// POUs/Functions/Gauges/Interfaces/FB_Gauge_Interface
(* This function block is created for interface devices between different PLC*)
(* Not all the Variables in the original structure is required, just few signals *)
(* They have to be linked to the custom created variables on the EL6692/5 primary side*)
FUNCTION_BLOCK FB_Gauge_Interface
VAR_INPUT
END_VAR
VAR_OUTPUT
	{attribute 'pytmc' := 'pv:'}
	VG : ST_VG;
END_VAR
VAR
	i_rPRESS AT%I*: REAL;  
	i_xAT_VAC AT%I*: BOOL;
	i_xPRESS_OK AT%I*: BOOL;
	
END_VAR

(* This function block is created for interface devices between different PLC*)
(* Not all the Variables in the original structure is required, just few signals *)
(* They have to be linked to the custom created variables on the EL6692/5 primary side*)

VG.rPRESS := i_rPRESS;
VG.xAT_VAC := i_xAT_VAC;
VG.xPRESS_OK := i_xPRESS_OK;

END_FUNCTION_BLOCK

// POUs/Functions/Gauges/Interfaces/FB_GaugeModbus
FUNCTION_BLOCK FB_GaugeModbus EXTENDS FB_GaugeBase
VAR_INPUT
	IP: STRING;	//IP of Legacy PLC
    nMBAddr	:WORD; //Start address of the Register Memory
	iBitOffset:INT :=0; // must be smaller than 32
	tTimeout :TIME:= T#1s;
END_VAR
VAR_OUTPUT
	VG: ST_VG;
	xNoPLCResponse: BOOL;
END_VAR
VAR
	fbPLCInputCoilsRx	:	FB_MBReadInputs;// (Modbus function 2)
	i_PLC_nBits	:	ARRAY [1..4] OF BYTE;
	ftReset	: F_TRIG; 
	tonRetry : TON;
	ErrCount:INT :=0;
	iIndex :INT;
	iBit:INT;
END_VAR
VAR CONSTANT
    nZero : INT := 0;
	nOne : INT := 1;
	nTwo : INT := 2;
	nThree : INT := 3;
	nFour : INT := 4;
	nFive : INT := 5;
	nSix : INT := 6;
	nSeven : INT := 7;
END_VAR

A_ReadMB();

ACTION A_ReadMB:
(*Credit to Alex Wallace*)
(* Modbus Info for Koyo
Modbus Addresses for
Koyo DL05/06/240/250/260/430/440/450 PLCs
PLC Memory Type		| Modbus start address Decimal (octal) | Function codes
Inputs (X)			  2048 (04000)							2
Special Relays (SP)	  3072 (06000)							2
Outputs (Y)			  2048 (04000)							1, 5, 15
Control Relays (C)	  3072 (06000)							1, 5, 15
Timer Contacts (T)	  6144 (014000)							1, 5, 15
Counter Contacts (CT) 6400 (014400)							1, 5, 15
Stage Status Bits (S) 6144 (012000)							1, 5, 15
*)

// Retry after some time
tonRetry.IN := NOT fbPLCInputCoilsRx.bBusy;
tonRetry.PT := T#10S;
tonRetry();

ftReset(CLK:=fbPLCInputCoilsRx.bBusy);
fbPLCInputCoilsRx.bExecute := ftReset.Q OR tonRetry.Q;

fbPLCInputCoilsRx(sIPAddr:=IP, nTCPPort:=502, nQuantity:=32, nMBAddr:=nMBAddr, cbLength:=SIZEOF(i_PLC_nBits),  pDestAddr:=ADR(i_PLC_nBits), tTimeout:=tTimeout);
//if there's a modbus error, set all incoming bits to zero
IF fbPLCInputCoilsRx.bError THEN
	i_PLC_nBits[1].0 := 0;
	i_PLC_nBits[1].1 := 0;
	i_PLC_nBits[1].2 := 0;
	i_PLC_nBits[1].3 := 0;
	i_PLC_nBits[1].4 := 0;
	i_PLC_nBits[1].5 := 0;
	i_PLC_nBits[1].6 := 0;
	i_PLC_nBits[1].7 := 0;
	i_PLC_nBits[2].0 := 0;
	i_PLC_nBits[2].1 := 0;
	i_PLC_nBits[2].2 := 0;
	i_PLC_nBits[2].3 := 0;
	i_PLC_nBits[2].4 := 0;
	i_PLC_nBits[2].5 := 0;
	i_PLC_nBits[2].6 := 0;
	i_PLC_nBits[2].7 := 0;
	VG.xPRESS_OK := FALSE;
	xNoPLCResponse:= TRUE;	
ELSIF NOT ftReset.Q AND fbPLCInputCoilsRx.cbRead > 0 THEN
	xNoPLCResponse:= FALSE;
	VG.rPRESS := 1E-8;
	iIndex:= REAL_TO_INT(iBitOffset/8);
	iBit:= (24 MOD 10);
	VG.xPRESS_OK := M_GetBit(iIndex,iBit);
	fbPLCInputCoilsRx.bExecute :=False;
ELSIF (*ftReset.Q*) NOT (fbPLCInputCoilsRx.bExecute) AND fbPLCInputCoilsRx.cbRead = 0 THEN
	xNoPLCResponse:= TRUE;		
END_IF

// Log Action
tAction(CLK:=   fbPLCInputCoilsRx.bError or xNoPLCResponse);
IF tAction.Q THEN 
ErrCount:= ErrCount+1; 
fbLogger(sMsg:='Modbus read error', eSevr:=TcEventSeverity.Critical);
END_IF
END_ACTION

METHOD M_GetBit : BOOL
VAR_INPUT
	iIndex:INT;
	iBit:INT;
END_VAR
Case iBit OF
	nZero: 
		M_GetBit:=i_PLC_nBits[iIndex].nZero;
	nOne: 
		M_GetBit:=i_PLC_nBits[iIndex].nOne;
	nTwo: 
		M_GetBit:=i_PLC_nBits[iIndex].nTwo;
	nThree: 
		M_GetBit:=i_PLC_nBits[iIndex].nThree;
	nFour: 
		M_GetBit:=i_PLC_nBits[iIndex].nFour;
	nFive: 
		M_GetBit:=i_PLC_nBits[iIndex].nFive;
	nSix: 
		M_GetBit:=i_PLC_nBits[iIndex].nSix;
	nSeven: 
		M_GetBit:=i_PLC_nBits[iIndex].nSeven;
END_CASE
END_METHOD

END_FUNCTION_BLOCK

// POUs/Functions/Gauges/Interfaces/FB_TGCC_ADS
(* This function block is created for interface devices between different PLC*)
(* Not all the Variables in the original structure is required, just few signals *)
(* The variable values are read via ADS using the symbol name*)
FUNCTION_BLOCK FB_TGCC_ADS Extends FB_ADS
VAR_INPUT
	sNetId : String; //NetID of the Destination PLC controller
	nPort : uint; // port number
	sVarName : string;// the variable name of the declared gauge function block.
	iWatchdog:UDINT;//The watchdog variable name written to by the remote plc
END_VAR
VAR_OUTPUT
	{attribute 'pytmc' := 'pv:'}
	IG : ST_VG;
	bError: BOOL;
END_VAR
VAR
	fb_CheckWatchdog: FB_CheckWatchdog;
	fb_Read_VG: FB_ReadAdsSymByName;
	ftReset: F_TRIG;
	xFirstPass: BOOL:= true;
END_VAR


ftReset(CLK:= fb_Read_VG.bBusy OR xFirstPass);
xFirstPass := false;
(*calling ADS read function*)

//IG.xPRESS_OK := false;	

fb_Read_VG(
	bRead:=ftReset.Q , 
	sNetId:= sNetId, 
	nPort:= nPort, 
	sVarName:= CONCAT(sVarName,'.IG'), 
	nDestAddr:= ADR(IG), 
	nLen:= SIZEOF(IG), 
	tTimeout:= , 
	eComMode:=eAdsComModeFastCom , 
	bBusy=> , 
	bError=> , 
	nErrorId=> );	
	

(*Error*)
fb_CheckWatchdog(
	bEnable:= TRUE, 
	tWatchdogTime:= T#900ms, 
	nCnt:= iWatchdog , 
	bWatchdog=> , 
	nLastCnt=> );
	
bError:= fb_Read_VG.bError OR fb_CheckWatchdog.bWatchdog;
tErrorPresent(CLK:=bError);

IF (fb_Read_VG.bError OR fb_CheckWatchdog.bWatchdog) THEN
IG.xPRESS_OK := FALSE;
END_IF;

(*Logger*)
ACT_Logger();

ACTION ACT_Logger:
IF tErrorPresent.Q THEN
 IF(fb_Read_VG.bError) THEN fbLogger(sMsg:='ADS Read Error', eSevr:=TcEventSeverity.Critical); END_IF;
 IF(fb_CheckWatchdog.bWatchdog) THEN fbLogger(sMsg:='ADS Watchdog Error', eSevr:=TcEventSeverity.Critical); END_IF;
END_IF
END_ACTION

END_FUNCTION_BLOCK

// POUs/Functions/Gauges/FB_972
{attribute 'no_check'}
FUNCTION_BLOCK FB_972  EXTENDS FB_GaugeBase
VAR_INPUT
END_VAR
VAR_OUTPUT
	{attribute 'pytmc' := '
    pv: 
	'}
	PG	: ST_VG;
END_VAR
VAR_IN_OUT
	
END_VAR
VAR
	rV : REAL;
	iTermBits: UINT := 32767 ; // The terminal's maximum value in bits
	(*IO*)
	i_iPRESS_R AT%I* :INT; // input Pressure // Link to analog Input
END_VAR

(* Standard MKS 9XX series conversion *)
(* works for 972 and 925 *)
// no div by zero
If (iTermBits=0) THEN iTermBits := 32767;END_IF
rV := 10*INT_TO_REAL(PG.i_iPRESS_R)/iTermBits;

IF rV > 1 THEN
	PG.rPRESS := LREAL_TO_REAL(EXPT(10, 2*rV-11));
	PG.xPRESS_OK := TRUE;
	PG.eState := Valid; //Press OK
ELSE
	PG.xPRESS_OK := FALSE;
	PG.eState := OoR;
END_IF



(* Soft IO Mapping*)
ACT_IO();

ACTION ACT_IO:
PG.i_iPRESS_R :=i_iPRESS_R;
END_ACTION

METHOD M_SetBits : BOOL
VAR_INPUT
	TermBits : UINT; // The terminal's maximum value in bits
END_VAR
This^.iTermBits := TermBits;
END_METHOD

END_FUNCTION_BLOCK

// POUs/Functions/Gauges/FB_9XX
(* Standard MKS 9XX series conversion *)
(* works for 925 *)
FUNCTION_BLOCK FB_9XX EXTENDS FB_GaugeBase
VAR_INPUT
END_VAR
VAR_OUTPUT
	{attribute 'pytmc' := '
    pv: 
	'}
	PG	: ST_VG;
END_VAR
VAR_IN_OUT
END_VAR
VAR
	rV : REAL;
	fbGaugeState : FB_PressureState;
	rMaxPressure	:	REAL := 760; //Torr
	rMinPressure	:	REAL := 1E-5; //Torr
	(*Default set point 50 mT*)
	rVAC_SP: REAL := 5E-2;
	iTermBits: UINT := 30518 ; // The terminal's maximum value in bits default el3174 as per vacuum architecture
	(*IO*)
	i_iPRESS_R AT%I* :INT; // input Pressure // Link to analog Input
END_VAR

(* Standard MKS 9XX series conversion *)
(* works for 972 and 925 *)

//Default setpoint 50 mT
IF PG.rVAC_SP = 0 THEN
	PG.rVAC_SP := rVAC_SP;
END_IF
// check no div by zero
If (iTermBits=0) THEN iTermBits := 30518;END_IF
rV := 10*INT_TO_REAL(PG.i_iPRESS_R)/iTermBits;

IF rV >= 0.99 THEN
	IF rV >= 0.99 AND rV <= 1 THEN
		PG.rPRESS := 1E-5;
	ELSE
		PG.rPRESS := LREAL_TO_REAL(EXPT(10, rV-6));
	END_IF
	PG.xPRESS_OK := TRUE;
	PG.eState := Valid;
ELSE
	PG.xPRESS_OK := FALSE;
	IF (rV = 0) THEN PG.eState := GaugeDisconnected;
		ELSE  PG.eState := PressInvalid;
	END_IF
END_IF

(* Setpoint evaluation *)
PG.xAT_VAC := PG.xPRESS_OK AND (PG.rPRESS < PG.rVAC_SP);


(*Logger*)
ACT_Logger();
(*Soft IO Mapping*)
ACT_IO();

ACTION ACT_IO:
PG.i_iPRESS_R :=i_iPRESS_R;
END_ACTION

ACTION ACT_Logger:

//STATE Logger  
IF ePrevState <> PG.eState THEN
	  CASE PG.eState OF
		ValidHi:
			fbLogger(sMsg:='Gauge pressure valid high.', eSevr:=TcEventSeverity.Info);
		ValidLo:
			fbLogger(sMsg:='Gauge pressure valid low.', eSevr:=TcEventSeverity.Info);
		Valid:
			fbLogger(sMsg:='Gauge pressure valid.', eSevr:=TcEventSeverity.Info);
  		GaugeDisconnected:
			fbLogger(sMsg:='Gauge Disconnected.', eSevr:=TcEventSeverity.Critical);
		PressInvalid:
			fbLogger(sMsg:='Gauge pressure invalid.', eSevr:=TcEventSeverity.Warning);
		OoR:
			fbLogger(sMsg:='Gauge pressure out of range.', eSevr:=TcEventSeverity.Warning);
		Starting:
			fbLogger(sMsg:='Gauge starting.', eSevr:=TcEventSeverity.Info);
	  END_CASE
	  ePrevState := PG.eState;  
  END_IF
END_ACTION

METHOD M_SetBits : BOOL
VAR_INPUT
	TermBits : UINT; // The terminal's maximum value in bits
END_VAR
This^.iTermBits := TermBits;
END_METHOD

END_FUNCTION_BLOCK

// POUs/Functions/Gauges/FB_CMR362
(* For Pfeiffer CMR 362 *)
FUNCTION_BLOCK FB_CMR362
VAR_INPUT
END_VAR
VAR_OUTPUT
		{attribute 'pytmc' := 'pv:'}
		PG : ST_VG;
END_VAR
VAR
	MinPressure: REAL := 7.5E-3; //Torr
	FullScale : REAL := 75.0 ; //Torr
	V : REAL;
	iTermBits: UINT := 32767 ; // The terminal's maximum value in bits
	(*IO*)
	i_iPRESS_R AT%I* :INT; // input Pressure // Link to analog Input
END_VAR


(* For Pfeiffer CMR 362 *)
(*Soft IO Mapping*)
ACT_IO();

(* Real-value calculation *)
If (iTermBits=0) THEN iTermBits := 32767;END_IF
V := 10*INT_TO_REAL(PG.i_iPRESS_R)/iTermBits;
	

IF V < 0.4 THEN

	PG.eState := GaugeDisconnected; //Most likely not connected

ELSIF V >= 0.4 AND V <= 1.0 THEN
	PG.rPRESS := MinPressure;
	PG.eState := ValidLo;

ELSIF V > 1 AND V <= 9.8 THEN

	PG.rPRESS := LREAL_TO_REAL((V-1)*0.125*FullScale);
	PG.eState := Valid;

ELSE
	
PG.eState := OoR; //Larger voltage, probably out of range?

END_IF


(* Pressure OK check *)
PG.xPRESS_OK := (PG.rPRESS >= MinPressure);

(*Soft IO Mapping*)
ACT_IO();

ACTION ACT_IO:
PG.i_iPRESS_R :=i_iPRESS_R;
END_ACTION

METHOD M_SetBits : BOOL
VAR_INPUT
	TermBits : UINT; // The terminal's maximum value in bits
END_VAR
This^.iTermBits := TermBits;
END_METHOD

END_FUNCTION_BLOCK

// POUs/Functions/Gauges/FB_GCM
(* For Baratron Pressure Gauge *)
(*The full-scale pressure times the ratio of the meas.
voltage to full-scale voltage (10V).
The minimum pressure is always going to be 5e-4 * F.S.V.*)
FUNCTION_BLOCK FB_GCM
VAR_IN_OUT

END_VAR
VAR_OUTPUT
	{attribute 'pytmc' := 'pv:'}
	PG	:	ST_VG;
END_VAR
VAR_INPUT
	i_rFULL_SCALE : REAL;
END_VAR
VAR
	rMinPressure: REAL;
	rHYST_PERC	:	REAL := 0.80;	// Hysteresis percentage
	rV	:REAL;
	iTermBits: UINT := 32767 ; // The terminal's maximum value in bits
	(*IO*)
	i_iPRESS_R AT%I* :INT; // input Pressure // Link to analog Input
END_VAR

(* Baratron Pressure Calc 
A. Wallace
2016-6-16
The full-scale pressure times the ratio of the meas.
voltage to full-scale voltage (10V).
The minimum pressure is always going to be 5e-4 * F.S.V.*)
PG.rFULL_SCALE := i_rFULL_SCALE;
rMinPressure := PG.rFULL_SCALE * 5E-4;

If (iTermBits=0) THEN iTermBits := 32767;END_IF
rV :=MAX((10*INT_TO_REAL(PG.i_iPRESS_R)/iTermBits),0);

PG.rPRESS := (PG.rFULL_SCALE/10)*rV;
IF PG.rPRESS > (rMinPressure)THEN
	PG.xPRESS_OK := TRUE;
ELSE
	PG.xPRESS_OK := FALSE;
END_IF

(*IO soft linking*)
ACT_IO();

ACTION ACT_IO:
PG.i_iPRESS_R :=i_iPRESS_R;
END_ACTION

METHOD M_SetBits : BOOL
VAR_INPUT
	TermBits : UINT; // The terminal's maximum value in bits
END_VAR
This^.iTermBits := TermBits;
END_METHOD

END_FUNCTION_BLOCK

// POUs/Functions/Gauges/FB_ITR90
(* This function block implements the Oerlikon Leybold IONVAC Hot Cathode ITR 90*)
FUNCTION_BLOCK FB_ITR90
VAR_INPUT
END_VAR
VAR_OUTPUT
	{attribute 'pytmc' := '
    pv: 
	'}
	PG : ST_VG;
END_VAR
VAR
	rV : REAL;	// input voltage
	rC: REAL := -0.125; // a constant in the manual (pressure unit dependent)
	rK: REAL := 1.0;// Calibration factor C (gas type dependent)
	iTermBits: UINT := 32767 ; // The terminal's maximum value in bits
	(*IO*)
	i_iPRESS_R AT%I* :INT; // input Pressure // Link to analog Input
END_VAR

(* This function block implements the Oerlikon Leybold IONVAC Hot Cathode ITR 90*)

(* Real-value calculation *)

rV := 10*INT_TO_REAL(PG.i_iPRESS_R)/iTermBits;	
PG.rPRESS := (LREAL_TO_REAL(EXPT(10,(rV-7.75)/0.75+rC))) * rK;


(* Pressure gauge State checks *)

//IF (rV <=9.7 ) AND (rV>=1) THEN
	//PG.eState := Valid; // normal
IF rV >= 0.5 AND rV <= 4.5 THEN
	PG.eState := ValidLo; //LO
ELSIF rV > 4.5 AND rV<= 9.9 THEN
	PG.eState := ValidHi; //HIGH
ELSIF rV < 0.5 THEN
	PG.eState := GaugeDisconnected; //not on
ELSE
	PG.eState := PressInvalid; //other fault - could be no gauge, controller powering up etc
END_IF



(* Pressure gauge OK checks *)
PG.xPRESS_OK := (rV <=9.9 ) AND (rV>=0.5);


(* Setpoint evaluation *)
PG.xAT_VAC := PG.xPRESS_OK AND PG.rPRESS < PG.rVAC_SP;


(*Soft IO Linking*)
ACT_IO();

ACTION ACT_IO:
PG.i_iPRESS_R :=i_iPRESS_R;
END_ACTION

METHOD M_SetBits : BOOL
VAR_INPUT
	TermBits : UINT; // The terminal's maximum value in bits
END_VAR
If (iTermBits=0) THEN iTermBits := 32767;END_IF
This^.iTermBits := TermBits;
END_METHOD

END_FUNCTION_BLOCK

// POUs/Functions/Gauges/FB_MKS_937A
(* 937A Logarithmic Output Conversion *)
(* 7-15-2015 *)
(* This function will read the pressure from any gauge on a 937A. *)
(* To be used when the specific device function block is not available *)
FUNCTION_BLOCK FB_MKS_937A
VAR_IN_OUT
	
END_VAR
VAR_INPUT
	PG	:	ST_VG := g_DummyVG; // Gauge Structure used to Interlock the ion gauges
END_VAR
VAR_OUTPUT
	{attribute 'pytmc' := 'pv: '}
	VG : ST_VG; // Vacuum Gauge Data Structure
END_VAR
VAR
	rV	:	REAL;
		(*IOs to be linked*)
	/// Controls and I/Os
	i_iPRESS_R AT %I* :INT; // input Pressure // Link to analog Input
	q_xHV_DIS AT %Q* : BOOL; // Disable Gauge High Voltage when True // 'TcLinkTo' (EL2794) ^Output
	
END_VAR

(* 937A Logarithmic Output Conversion *)
(* 7-15-2015 *)
(* This function will read the pressure from any gauge on a 937A. *)

rV := 10*INT_TO_REAL(VG.i_iPRESS_R)/32767;
VG.rPRESS := LREAL_TO_REAL(EXPT(10,rV/0.6-12));


(* Ion Gauge Protection Functions *)
(* If the PG pressure is greater than the VG.PRO_SP then the gauge is disabled *)
(* If the PG pressure is less than the VG.PRO_SP then the gauge is enabled *)
(* This FB also implements some hysteresis so the gauge doesn't have rapid power cycling while near the turn on boundary *)

IF PG.rPRESS < VG.rPRO_SP THEN

VG.q_xHV_DIS :=  NOT VG.xHV_SW;

ELSIF NOT VG.q_xHV_DIS THEN
	IF VG.rPRESS > VG.rPRO_SP + VG.rHYS_PR OR PG.rPRESS > VG.rPRO_SP + VG.rHYS_PR THEN
		VG.q_xHV_DIS := TRUE;
	END_IF
ELSE
	VG.q_xHV_DIS := TRUE;
END_IF


(* Pressure gauge OK checks *)
VG.xPRESS_OK := (rV <=9.6 ) AND (rV>=0.6); //legacy

IF (rV <=9.6 ) AND (rV>=0.6) THEN
	VG.eState := Valid; // normal
ELSIF rV >= 0.18 AND rV <= 0.22 THEN
	VG.eState := ValidLo; //LO
ELSIF rV >= 9.7 AND rV<= 9.9 THEN
	VG.eState := ValidHi; //HIGH
ELSIF rV < 0.18 THEN
	VG.eState := GaugeDisconnected; //not on
ELSE
	VG.eState := PressInvalid; //other fault - could be no gauge, controller powering up etc
END_IF

(* Setpoint evaluation *)
VG.xAT_VAC := (VG.eState =Valid) AND VG.rPRESS < VG.rVAC_SP;

(*Soft IO Linking*)
ACT_IO();

ACTION ACT_IO:
(*soft link inputs*)
VG.i_iPRESS_R:=	i_iPRESS_R; 

(*soft link outputs*)
q_xHV_DIS := VG.q_xHV_DIS;
END_ACTION

END_FUNCTION_BLOCK

// POUs/Functions/Gauges/FB_MKS_937B
(* 937B Logarithmic Output Conversion *)
(* 5-20-2016, Alex Wallace and Scott Stubbs *)
(* This function will read the pressure from any gauge on a 937B. *)
(* To be used when the specific device function block is not available *)
FUNCTION_BLOCK FB_MKS_937B
VAR_IN_OUT
			
END_VAR
VAR_INPUT
	PG	:	ST_VG := g_DummyVG; // Gauge Structure used to Interlock the ion gauges
END_VAR
VAR_OUTPUT
	{attribute 'pytmc' := 'pv: '}
	VG : ST_VG; // Vacuum Gauge Data Structure
	
	

END_VAR
VAR
	rV	:	REAL;
	
	
		(*IOs to be linked*)
	/// Controls and I/Os
	i_iPRESS_R AT %I* :INT; // input Pressure // Link to analog Input
	q_xHV_DIS AT %Q* : BOOL; // Disable Gauge High Voltage when True // 'TcLinkTo' (EL2794) ^Output
	
END_VAR

(* 937B Logarithmic Output Conversion *)
(* 5-20-2016, Alex Wallace and Scott Stubbs *)
(* This function will read the pressure from any gauge on a 937B. *)

rV := 10*INT_TO_REAL(VG.i_iPRESS_R)/32767;
VG.rPRESS := LREAL_TO_REAL(EXPT(10,(rV-7.2)/0.6));


(* Gauge Protection Functions *)
(* If the PG pressure is greater than the VG.PRO_SP then the gauge is disabled *)
(* If the PG pressure is less than the VG.PRO_SP then the gauge is enabled *)
(* This FB also implements some hysteresis so the gauge doesn't have rapid power cycling while near the turn on boundary *)

IF PG.rPRESS < VG.rPRO_SP THEN // might enable the gauge automatically, do we want that?

VG.q_xHV_DIS := NOT VG.xHV_SW;

ELSIF NOT VG.q_xHV_DIS THEN
	IF VG.rPRESS > VG.rPRO_SP + VG.rHYS_PR OR PG.rPRESS > VG.rPRO_SP + VG.rHYS_PR THEN
		VG.q_xHV_DIS := TRUE;
	END_IF
ELSE
	VG.q_xHV_DIS := TRUE;
END_IF


(* Pressure gauge OK checks *)
VG.xPRESS_OK := (rV <=9.6 ) AND (rV>=0.6);
(* Pressure gauge State checks *)
IF (rV <=9.7 ) AND (rV>=0.6) THEN
	VG.eState := Valid; // normal
ELSIF rV >= 0.18 AND rV <= 0.22 THEN
	VG.eState := ValidLo; //LO
ELSIF rV > 9.7 AND rV<= 9.9 THEN
	VG.eState := ValidHi; //HIGH
ELSIF rV < 0.18 THEN
	VG.eState := GaugeDisconnected; //not on
ELSE
	VG.eState := PressInvalid; //other fault - could be no gauge, controller powering up etc
END_IF

(* Setpoint evaluation *)
VG.xAT_VAC := (VG.eState =Valid) AND VG.rPRESS < VG.rVAC_SP;


(*Soft IO Linking*)
// check ethercat Diagnostics
ACT_IO();

ACTION ACT_IO:
(*soft link inputs*)
VG.i_iPRESS_R:=	i_iPRESS_R; 

(*soft link outputs*)
q_xHV_DIS := VG.q_xHV_DIS;
END_ACTION

END_FUNCTION_BLOCK

// POUs/Functions/Gauges/FB_MKS275
(* This function block is used to provide protection and automatic turn on of ion gauges,
 it also manages the turn on of the AT_VAC boolean, and checks to make sure the pressure is good *)
(* For MKS 275 mini-convectron *)
{attribute 'no_check'}
FUNCTION_BLOCK FB_MKS275 EXTENDS FB_GaugeBase
VAR_IN_OUT

END_VAR
VAR_INPUT
END_VAR

VAR_OUTPUT
	{attribute 'pytmc' := '
    pv: 
	'}
	PG : ST_VG;
END_VAR
VAR
	V : REAL;
	iTermBits: UINT := 32767 ; // The terminal's maximum value in bits
	Vlowest: REAL := 10;
	(*IO*)
	i_iPRESS_R AT%I* :INT; // input Pressure // Link to analog Input
END_VAR

VAR CONSTANT
	MinPressure: REAL := 1E-4;
	rDeadband : REAL :=0.05;
	rValidLoBoundary	:	REAL := 0.375; //  0.375V as per manual page 27
	rValidHiBoundary	:	REAL := 5.659;// 5.534; // manual page 27
	rDisconnectedBoundary	:	REAL := 0.3;
END_VAR

(* This function block is used to provide protection and automatic turn on of ion gauges,
 it also manages the turn on of the AT_VAC boolean, and checks to make sure the pressure is good *)
(* For MKS 275 mini-convectron *)

//Default setpoint 50 mT
IF PG.rVAC_SP = 0 THEN
	PG.rVAC_SP := 5E-2;
END_IF

(* Real-value calculation *)
If (iTermBits=0) THEN iTermBits := 32767;END_IF
V := 10*INT_TO_REAL(PG.i_iPRESS_R)/iTermBits;	

Vlowest := MIN(V, Vlowest);

IF V > rDisconnectedBoundary AND V < rValidLoBoundary  THEN
	PG.rPRESS := MinPressure;
	PG.eState := ValidLo;
	
ELSIF V >= rValidLoBoundary AND V < rValidLoBoundary +rDeadband  THEN
	PG.rPRESS := MAX( MinPressure, LREAL_TO_REAL( -0.02585 + 0.03767*V + 0.04563*EXPT(V,2)+ 0.1151*EXPT(V,3) - 0.04158*EXPT(V,4)+ 0.008737*EXPT(V,5)) );
	PG.eState := ValidLo;
	
ELSIF V >= rValidLoBoundary AND V < 2.842 THEN
	PG.rPRESS := MAX( MinPressure, LREAL_TO_REAL( -0.02585 + 0.03767*V + 0.04563*EXPT(V,2)+ 0.1151*EXPT(V,3) - 0.04158*EXPT(V,4)+ 0.008737*EXPT(V,5)) );
	PG.eState := Valid;

ELSIF V >= 2.842 AND V < 4.945 THEN
	PG.rPRESS := LREAL_TO_REAL((0.1031-0.02322*V+0.07229*EXPT(V,2))/(1-0.3986*V+0.07438*EXPT(V,2)-0.006866*EXPT(V,3)));
	PG.eState := Valid;

ELSIF V >= 4.945 AND V < rValidHiBoundary THEN
	PG.rPRESS := LREAL_TO_REAL((100.624-20.5623*V)/(1-0.37679*V+0.0348656*EXPT(V,2)));
	PG.eState := ValidHi;

ELSIF V <= rDisconnectedBoundary THEN
	PG.eState := GaugeDisconnected; //Most likely not connected
	PG.rPRESS := -1;

ELSE
	PG.eState := OoR; //Larger voltage, probably out of range?
	PG.rPRESS := -1;
END_IF

(* Protection Functions *)
(* If the PG pressure is greater than the IG.PRO_SP then the gauge is disabled *)
(* If the PG pressure is less than the IG.PRO_SP then the gauge is enabled *)
(* This FB also implements some hysteresis so the gauge doesn't have rapid power cycling while near the turn on boundary *)

(* Pressure OK check *)
PG.xPRESS_OK := (PG.rPRESS >= MinPressure);

(* Setpoint evaluation *)
PG.xAT_VAC := PG.xPRESS_OK AND (PG.rPRESS<=PG.rVAC_SP);

(*Logger*)
ACT_Logger();

(*Soft IO Mapping *)
IO();

ACTION ACT_Logger:

//STATE Logger  
if (PG.xLog) THEN
	IF ePrevState <> PG.eState THEN
	  CASE PG.eState OF
		ValidHi:
			fbLogger(sMsg:='Gauge pressure valid high.', eSevr:=TcEventSeverity.Info);
		ValidLo:
			fbLogger(sMsg:='Gauge pressure valid low.', eSevr:=TcEventSeverity.Info);
		Valid:
			fbLogger(sMsg:='Gauge pressure valid.', eSevr:=TcEventSeverity.Info);
  		GaugeDisconnected:
			fbLogger(sMsg:='Gauge Disconnected.', eSevr:=TcEventSeverity.Critical);
		PressInvalid:
			fbLogger(sMsg:='Gauge pressure invalid.', eSevr:=TcEventSeverity.Warning);
		OoR:
			fbLogger(sMsg:='Gauge pressure out of range.', eSevr:=TcEventSeverity.Warning);
		Starting:
			fbLogger(sMsg:='Gauge starting.', eSevr:=TcEventSeverity.Info);
	  END_CASE
	  ePrevState := PG.eState;  
  END_IF 
END_IF
END_ACTION

ACTION IO:
PG.i_iPRESS_R :=i_iPRESS_R;
PG.sPath := sPath;
END_ACTION

METHOD M_SetBits : BOOL
VAR_INPUT
	TermBits : UINT; // The terminal's maximum value in bits
END_VAR
This^.iTermBits := TermBits;
END_METHOD

END_FUNCTION_BLOCK

// POUs/Functions/Gauges/FB_MKS317
(* This function is for the Pirani MKS 317 connected to a 937A/B *)
(* This function block is used to provide protection and automatic turn on of ion gauges,
 it also manages the turn on of the AT_VAC boolean, and checks to make sure the pressure is good *)

FUNCTION_BLOCK FB_MKS317 Extends FB_GaugeBase
VAR_IN_OUT
END_VAR
VAR_INPUT
	b937A :BOOL := FALSE; // True if this gauge is connected to MKS937A controller, False if connected to MKS937B controller
END_VAR
VAR_OUTPUT
	{attribute 'pytmc' := '
    pv: 
	'}
	PG : ST_VG;
END_VAR
VAR
	rV	:	REAL;

	(*IO*)
	i_iPRESS_R AT%I* :INT; // input Pressure // Link to analog Input
END_VAR

VAR CONSTANT
	rMinPressure: REAL := 1E-4;
	rDefaultVAC_SP: REAL :=5E-2; // Default 50 mT
	rDisconnectedBoundary	:	REAL := 0.10;
	rValidLoBoundary	:	REAL := 0.22;
	rValidBoundaryMin	:	REAL := 0.6;
	rValidHiBoundary	:	REAL := 9.7;
	rValidHiBoundaryMax	:	REAL := 9.9; 
	rNoSensorBoundary	:	REAL := 10;
END_VAR

(* 937B Logarithmic Output Conversion *)
(* 5-20-2016, Alex Wallace and Scott Stubbs *)
(* 09-28-2018, Margaret Ghaly *)
(* This function will read the pressure from any gauge on a 937B. *)

rV := 10*INT_TO_REAL(PG.i_iPRESS_R)/32767;
if (b937A) THEN
	PG.rPRESS := LREAL_TO_REAL(EXPT(10,((rV)/0.6)-12)); //manual page 61 MKS937A
	ELSE
	PG.rPRESS := LREAL_TO_REAL(EXPT(10,(rV-7.2)/0.6));	//manual page 73 MKS937B
END_IF


//Default setpoint 
IF PG.rVAC_SP = 0 THEN
	PG.rVAC_SP := rDefaultVAC_SP;
END_IF

IF (rV <=rValidHiBoundary ) AND (rV>=rValidBoundaryMin) THEN
	PG.eState := Valid; // normal
ELSIF rV >= rDisconnectedBoundary AND rV <= rValidLoBoundary THEN
	PG.eState := ValidLo; //LO
	PG.rPRESS := rMinPressure;
ELSIF rV > rValidHiBoundary AND rV<= rValidHiBoundaryMax THEN
	PG.eState := ValidHi; //HIGH
ELSIF rV < rDisconnectedBoundary THEN
	PG.eState := GaugeDisconnected; //not on
	PG.rPRESS := -1;
ELSE
	PG.eState := PressInvalid; //other fault - could be no gauge, controller powering up etc
	PG.rPRESS := -1;
END_IF

(* Pressure OK check *)
(* Pressure gauge OK checks *)
PG.xPRESS_OK := (rV <=rValidHiBoundary ) AND (rV>=rDisconnectedBoundary);
//PG.xPRESS_OK := (PG.rPRESS >= rMinPressure);

(* Setpoint evaluation *)
PG.xAT_VAC := (*(PG.eState =Valid)*) PG.xPRESS_OK AND PG.rPRESS <= PG.rVAC_SP;

(*Logger*)
ACT_Logger();

(*soft io*)
IO();

ACTION ACT_Logger:

//STATE Logger  
IF (PG.xLog) THEN
	IF ePrevState <> PG.eState THEN
		  CASE PG.eState OF
			ValidHi:
				fbLogger(sMsg:='Gauge pressure valid high.', eSevr:=TcEventSeverity.Info);
			ValidLo:
				fbLogger(sMsg:='Gauge pressure valid low.', eSevr:=TcEventSeverity.Info);
			Valid:
				fbLogger(sMsg:='Gauge pressure valid.', eSevr:=TcEventSeverity.Info);
			GaugeDisconnected:
				fbLogger(sMsg:='Gauge Disconnected.', eSevr:=TcEventSeverity.Critical);
			PressInvalid:
				fbLogger(sMsg:='Gauge pressure invalid.', eSevr:=TcEventSeverity.Warning);
			OoR:
				fbLogger(sMsg:='Gauge pressure out of range.', eSevr:=TcEventSeverity.Warning);
			Starting:
				fbLogger(sMsg:='Gauge starting.', eSevr:=TcEventSeverity.Info);
		  END_CASE
		  ePrevState := PG.eState;  
	  END_IF
 END_IF
END_ACTION

ACTION IO:
PG.i_iPRESS_R :=i_iPRESS_R;

PG.sPath := sPath;
END_ACTION

END_FUNCTION_BLOCK

// POUs/Functions/Gauges/FB_MKS392
(* This function block implements the MKS392 gauge*)
FUNCTION_BLOCK FB_MKS392
VAR_INPUT
END_VAR
VAR_OUTPUT
	{attribute 'pytmc' := '
    pv: 
	'}
	PG : ST_VG;
END_VAR
VAR
	rV : REAL;	// input voltage
	iTermBits: UINT := 32767 ; // The terminal's maximum value in bits
	(*IO*)
	i_iPRESS_R AT%I* :INT; // input Pressure // Link to analog Input
END_VAR

(* Real-value calculation *)
rV := 10*INT_TO_REAL(PG.i_iPRESS_R)/iTermBits;	
PG.rPRESS := (LREAL_TO_REAL(EXPT(10,(2*rV)-11)));


(* Pressure gauge State checks *)

IF rV >= 0.5 AND rV <= 3.5 THEN
	PG.eState := ValidLo; //LO
ELSIF rV > 3.5 AND rV<= 6.5 THEN
	PG.eState := ValidHi; //HIGH
ELSIF rV < 0.5 THEN
	PG.eState := GaugeDisconnected; //not on
ELSE
	PG.eState := PressInvalid; //other fault - could be no gauge, controller powering up etc
END_IF



(* Pressure gauge OK checks *)
PG.xPRESS_OK := (rV <=6.5 ) AND (rV>=0.5);


(* Setpoint evaluation *)
PG.xAT_VAC := PG.xPRESS_OK AND PG.rPRESS < PG.rVAC_SP;


(*Soft IO Linking*)
ACT_IO();

ACTION ACT_IO:
PG.i_iPRESS_R :=i_iPRESS_R;
END_ACTION

END_FUNCTION_BLOCK

// POUs/Functions/Gauges/FB_MKS422
(* This function is for the Cold Cathode MKS 422 connected to a 937A/B *)
(*This function provides ILK and Set Point Protection for the Cold Cathode*)
FUNCTION_BLOCK FB_MKS422 EXTENDS FB_GaugeBase
VAR_IN_OUT
		
END_VAR
VAR_INPUT
		PG	:	ST_VG; // Pirani Gauge Structure used to Interlock the Cold Cathode
		b937A :BOOL:=FALSE; // True if this gauge is connected to MKS937A controller, False if connected to MKS937B controller
END_VAR
VAR_OUTPUT
	{attribute 'pytmc' := '
    pv: 
	'}
	IG : ST_VG; // The Cold Cathode Data Structure
END_VAR
VAR
	rV	:	REAL;
	
	timer:TON;
	(*IOs to be linked*)
	/// Controls and I/Os
	i_iPRESS_R AT %I* :INT; // input Pressure // Link to analog Input
	q_xHV_DIS AT %Q* : BOOL := True; // Disable Gauge High Voltage when True // 'TcLinkTo' (EL2794) ^Output
END_VAR
VAR CONSTANT
	MinPressure: REAL := 1E-10;
	cDefaultPressure : REAL := 0;
END_VAR

(* 937B Logarithmic Output Conversion *)
(* 5-20-2016, Alex Wallace and Scott Stubbs *)
(* 09-28-2018, Margaret Ghaly *)
(* This function will read the pressure from any gauge on a 937B. *)

(*Soft IO Linking*)
IO();

(*Pressure readbacks*)
rV := 10*INT_TO_REAL(IG.i_iPRESS_R)/32767;
if (b937A) THEN
	IG.rPRESS := LREAL_TO_REAL(EXPT(10,((rV)/0.6)-12)); //manual page 61 MKS937A
	ELSE
	IG.rPRESS := LREAL_TO_REAL(EXPT(10,(rV-7.2)/0.6));	//manual page 73 MKS937B
END_IF

	

(* Pressure gauge State checks *)
IF (rV <=9.6 ) AND (rV>=0.6) THEN
	IG.eState := Valid; // normal
ELSIF rV >= 0.18 AND rV <= 0.22 THEN 
	IG.eState := ValidLo; //LO
ELSIF rV > 9.6 AND rV<= 9.9 THEN
	IG.eState := ValidHi; //HIGH
ELSIF rV < 0.18 THEN // 
	IG.eState := GaugeDisconnected; //not on
	IG.rPRESS :=cDefaultPressure;
ELSE
	IG.eState := PressInvalid; //other fault - could be no gauge, controller powering up etc
	IG.rPRESS :=cDefaultPressure;
END_IF


(* Ion Gauge Protection Functions *)
(* If the PG pressure is greater than the VG.PRO_SP then the gauge is disabled *)
(* If the PG pressure is less than the VG.PRO_SP then the gauge is enabled *)
(* This FB also implements some hysteresis so the gauge doesn't have rapid power cycling while near the turn on boundary *)

	IF (PG.rPRESS <= IG.rPRO_SP) THEN
		 IG.q_xHV_DIS := NOT IG.xHV_SW;
		 IG.xILKOk := TRUE;
	ELSIF NOT IG.q_xHV_DIS AND timer.Q THEN
		IF IG.rPRESS > (IG.rPRO_SP + IG.rHYS_PR) OR PG.rPRESS > (IG.rPRO_SP + IG.rHYS_PR) THEN
		IG.q_xHV_DIS := TRUE;
		IG.xHV_SW := FALSE;
		END_IF
	ELSE 
		IG.q_xHV_DIS := TRUE;
		IG.xHV_SW := FALSE;
		IG.xILKOk := FALSE;
 	END_IF
 


 
(* Pressure gauge OK checks *)
IG.xPRESS_OK := (rV <=9.6 ) AND (rV>=0.6);


(* Setpoint evaluation *)
IG.xAT_VAC := IG.xPRESS_OK AND IG.rPRESS < IG.rVAC_SP;


(*Logger*)
ACT_Logger();
(*Soft IO Linking*)
// check ethercat Diagnostics
IO();

timer(IN:= NOT IG.q_xHV_DIS, PT:= T#2s);

ACTION ACT_Logger:
// ILK logger
IF (IG.xLog) THEN
	IF NOT IG.xILKOk AND NOT IG.q_xHV_DIS THEN
			fbLogger(sMsg:='Lost external interlock while gauge was on.', eSevr:=TcEventSeverity.Critical);  	
	END_IF
	
	
	// Log Action
	tAction(CLK:=  IG.xHV_SW);
	IF tAction.Q THEN fbLogger(sMsg:='Ion gauge commanded to switch on', eSevr:=TcEventSeverity.Info); END_IF
	
	
	
	//STATE Logger  
	IF ePrevState <> IG.eState THEN
		  CASE IG.eState OF
			ValidHi:
				fbLogger(sMsg:='Gauge pressure valid high.', eSevr:=TcEventSeverity.Info);
			ValidLo:
				fbLogger(sMsg:='Gauge pressure valid low.', eSevr:=TcEventSeverity.Info);
			Valid:
				fbLogger(sMsg:='Gauge pressure valid.', eSevr:=TcEventSeverity.Info);
			GaugeDisconnected:
				fbLogger(sMsg:='Gauge Disconnected.', eSevr:=TcEventSeverity.Critical);
			PressInvalid:
				fbLogger(sMsg:='Gauge pressure invalid.', eSevr:=TcEventSeverity.Warning);
			OoR:
				fbLogger(sMsg:='Gauge pressure out of range.', eSevr:=TcEventSeverity.Warning);
			Starting:
				fbLogger(sMsg:='Gauge starting.', eSevr:=TcEventSeverity.Info);
		  END_CASE
		  ePrevState := IG.eState;  
	  END_IF
END_IF
END_ACTION

ACTION IO:
(*soft link inputs*)
IG.i_iPRESS_R:=	i_iPRESS_R; 

(*soft link outputs*)
q_xHV_DIS := IG.q_xHV_DIS;

IG.sPath := sPath;
END_ACTION

METHOD M_AutoOn : BOOL
VAR_INPUT
END_VAR
this^.IG.q_xHV_DIS:= FALSE;
END_METHOD

METHOD M_HVE : BOOL
VAR_INPUT
		enable:bool; // set to true to enable, false to disable;
END_VAR

this^.IG.xHV_SW:= (enable);
END_METHOD

END_FUNCTION_BLOCK

// POUs/Functions/Gauges/FB_MKS500
(* This function is for the Cold Cathode MKS 500. If connected to Beckhoff EP boxes.
Set the EP bit to TRUE, this is necessary for the MKS500-to-EP box interface beacuse the EP
boxes do not natively support the 5v IO signals on the MKS500 gauge.*)
(*This function provides ILK and Set Point Protection for the Cold Cathode*)
(* 500 Logarithmic Output Conversion, factory default configuration *)
FUNCTION_BLOCK FB_MKS500 EXTENDS FB_GaugeBase
VAR_IN_OUT
		
END_VAR
VAR_INPUT
	PG	:	ST_VG;
	bEP : BOOL :=FALSE; // Set to True if This Gauge is connected to EP BOX and not EL Terminals
END_VAR
VAR_OUTPUT
{attribute 'pytmc' := '
    pv: 
	'}
	IG : ST_VG;
END_VAR
VAR
	rV : REAL;
	GaugeTurnOnTmr : TON;
	iTermBits: UINT := 32767 ; // The terminal's maximum value in bits
	(*IOs to be linked*)
	/// Controls and I/Os
	i_iPRESS_R AT %I* :INT; // input Pressure // Link to analog Input
	q_xHV_DIS AT %Q* : BOOL; // Enable High Voltage when True // 'TcLinkTo' (EP2624) ^Output
	// only for EL and ES terminal
	i_xHV_ON AT %I*	: BOOL; //  True when High Voltage is on  // 'TcLinkTo' (EL1124) ^Input
	i_xDisc_Active AT %I* : BOOL;// Discharge Current Active // 'TcLinkTo' (EL1124) ^Input
	
END_VAR

VAR CONSTANT
	// Ranges has to match the configurator software
	pBase : REAL :=1.0E-10;//default curve base pressure is 1E-10. Confusing since can't actually read that low using analog out.
	vBase : REAL := 1;
	vDisconnected : REAL:= 0.5;
	vSlope : REAL := 1.0; 
	vGaugeOff: REAL := 9.8;
	vNoDischarge: REAL := 9.3;
	MinPressure: REAL := 1E-10;
	cDefaultPressure : REAL := 0;
	rDeadband : REAL :=0.3;
END_VAR

(* 500 Logarithmic Output Conversion, factory default configuration *)
If (iTermBits=0) THEN iTermBits := 32767;END_IF
rV := 10*INT_TO_REAL(IG.i_iPRESS_R)/iTermBits;

(* Set Guage State based on the Analog voltage*)
IF rV < vDisconnected THEN
	IG.eState := GaugeDisconnected;
	IG.rPRESS := cDefaultPressure;
ELSIF rV >= vDisconnected AND rV < (vNoDischarge -rDeadband)  THEN
	IG.eState := Valid;
	IG.rPRESS := LREAL_TO_REAL(EXPT(10,((rV-vBase)/vSlope+LOG(pBase))));
ELSIF rV >= (vNoDischarge -rDeadband) AND rV <(vGaugeOff -rDeadband)   THEN
	IG.eState := Starting;
	IG.rPRESS := LREAL_TO_REAL(EXPT(10,((rV-vBase)/vSlope+LOG(pBase))));
ELSIF rV >= (vGaugeOff -rDeadband) THEN
	IG.eState := Off;
	//IG.rPRESS := LREAL_TO_REAL(EXPT(10,((rV-vBase)/vSlope+LOG(pBase))));
	IG.rPRESS := cDefaultPressure;
ELSE
	IG.eState := OoR;
	//IG.rPRESS := LREAL_TO_REAL(EXPT(10,((rV-vBase)/vSlope+LOG(pBase))));
	IG.rPRESS := cDefaultPressure;
END_IF

(* Set Guage State based on the inputs HV ON and Discharge current*)
If (NOT bEP) THEN
	IF IG.i_xHV_ON AND NOT IG.i_xDisc_Active THEN
		IG.eState := Starting;
		IG.rPRESS := LREAL_TO_REAL(EXPT(10,((rV-vBase)/vSlope+LOG(pBase))));
	ELSIF IG.i_xHV_ON AND IG.i_xDisc_Active THEN
		IG.eState := Valid;
		IG.rPRESS := LREAL_TO_REAL(EXPT(10,((rV-vBase)/vSlope+LOG(pBase))));
	ELSIF NOT IG.i_xHV_ON AND NOT IG.i_xDisc_Active THEN
		IG.eState := Off;
		IG.rPRESS := cDefaultPressure;
	END_IF
END_IF

(* Ion Gauge Protection Functions *)
(* If the PG pressure is greater than the VG.PRO_SP then the gauge is disabled *)
(* If the PG pressure is less than the VG.PRO_SP then the gauge is enabled *)
(* This FB also implements some hysteresis so the gauge doesn't have rapid power cycling while near the turn on boundary *)


IF PG.rPRESS <= IG.rPRO_SP AND PG.xPRESS_OK THEN
	IG.q_xHV_DIS := IG.xHV_SW;
	IG.xILKOk := TRUE;
ELSIF IG.q_xHV_DIS THEN
	IF IG.rPRESS > (IG.rPRO_SP + IG.rHYS_PR)  OR PG.rPRESS > (IG.rPRO_SP + IG.rHYS_PR) THEN
		IG.q_xHV_DIS := FALSE;
		IG.xHV_SW := FALSE;
	END_IF
ELSE
	IG.q_xHV_DIS := FALSE;
	IG.xHV_SW := FALSE;
	IG.xILKOk := FALSE;
END_IF

(* Pressure gauge OK checks *)

GaugeTurnOnTmr(IN:=IG.q_xHV_DIS, PT:=T#10S, Q=>IG.xTurnOnTime);


//Backwards compatibility
IG.xPRESS_OK := (IG.eState = Valid) OR IG.xBAKEOUT;

(* Setpoint evaluation *)
IG.xAT_VAC := (IG.xPRESS_OK AND (IG.rPRESS < IG.rVAC_SP)) OR IG.xBAKEOUT AND (IG.eState = Valid) ;

ACT_Logger();
(*Soft IO Linking*)
// check ethercat Diagnostics
IO();

ACTION ACT_Logger:
// ILK logger
IF (IG.xLog) THEN
	IF NOT IG.xILKOk AND IG.q_xHV_DIS THEN
			fbLogger(sMsg:='Lost external interlock while gauge was on.', eSevr:=TcEventSeverity.Critical);  	
	END_IF
	
	
	// Log Action
	tAction(CLK:=   IG.xHV_SW);
	IF tAction.Q THEN fbLogger(sMsg:='Ion gauge commanded to switch on', eSevr:=TcEventSeverity.Info); END_IF
	
	
	
	//STATE Logger  
	tState(CLK:=  ePrevState <> IG.eState);
	IF ePrevState <> IG.eState THEN
		  CASE IG.eState OF
			ValidHi:
				fbLogger(sMsg:='Gauge pressure valid high.', eSevr:=TcEventSeverity.Info);
			ValidLo:
				fbLogger(sMsg:='Gauge pressure valid low.', eSevr:=TcEventSeverity.Info);
			Valid:
				fbLogger(sMsg:='Gauge pressure valid.', eSevr:=TcEventSeverity.Info);
			GaugeDisconnected:
				fbLogger(sMsg:='Gauge Disconnected.', eSevr:=TcEventSeverity.Critical);
			PressInvalid:
				fbLogger(sMsg:='Gauge pressure invalid.', eSevr:=TcEventSeverity.Warning);
			OoR:
				fbLogger(sMsg:='Gauge pressure out of range.', eSevr:=TcEventSeverity.Warning);
			Starting:
				fbLogger(sMsg:='Gauge starting.', eSevr:=TcEventSeverity.Info);
		  END_CASE
		  ePrevState := IG.eState;  
	  END_IF
END_IF
END_ACTION

ACTION IO:
(*soft link inputs*)
IG.i_iPRESS_R:=	i_iPRESS_R; 
IG.i_xHV_ON:= i_xHV_ON;
IG.i_xDisc_Active:=i_xDisc_Active; 
(*soft link outputs*)
q_xHV_DIS := IG.q_xHV_DIS;

IG.sPath := sPath;
END_ACTION

METHOD M_HVE : BOOL
VAR_INPUT
		enable:bool; // set to true to enable, false to disable;
END_VAR

this^.IG.xHV_SW:= enable;
END_METHOD

METHOD M_SetBits : BOOL
VAR_INPUT
	TermBits : UINT; // The terminal's maximum value in bits
END_VAR
This^.iTermBits := TermBits;
END_METHOD

END_FUNCTION_BLOCK

// POUs/Functions/Gauges/FB_MKS722
(* This function is for the MKS 722*)

FUNCTION_BLOCK FB_MKS722
VAR_IN_OUT
	
END_VAR
VAR_OUTPUT
	{attribute 'pytmc' := '
    pv: 
	'}
	VG	:	ST_VG;
END_VAR
VAR_INPUT
	i_rMinPressure	:	REAL;
	i_rMaxPressure	:	REAL;
END_VAR
VAR
	iTermBits: UINT := 32767 ; // The terminal's maximum value in bits
	rMinPressure: REAL;
	rVMin	:	REAL := 0.01; // Anything less than this voltage is considered disconnected
	rVMax :	REAL := 10.5; // Anything more than this is considered invalid
	rV	:REAL;
	
	(*IO*)
	i_iPRESS_R AT%I* :INT; // input Pressure // Link to analog Input
END_VAR



(* Real-value calculation *)
If (iTermBits=0) THEN iTermBits := 32767;END_IF
rV := 10*INT_TO_REAL(VG.i_iPRESS_R)/iTermBits;	


// Is the gauge plugged in, and within a reasonable range?
IF rV < rVMin THEN
	VG.eState := GaugeDisconnected;
ELSIF rV > rVMax THEN
	VG.eState := PressInvalid;
ELSIF VG.rPRESS >= rMinPressure AND VG.rPRESS <= i_rMaxPressure THEN
				VG.eState := Valid;
ELSIF VG.rPRESS < i_rMinPressure THEN
				VG.eState := ValidLo;
ELSE
				VG.eState := ValidHi;
END_IF
			
// Legacy Press OK boolean eval
VG.xPRESS_OK := VG.eState >= gc_GaugeValidState;

(*IO Soft Mapping*)
ACT_IO();

ACTION ACT_IO:
VG.i_iPRESS_R :=i_iPRESS_R;
END_ACTION

END_FUNCTION_BLOCK

// POUs/Functions/Gauges/FB_MKS909
(* Standard MKS 909 hot cathode *)
(* works for 972 and 925 *)

FUNCTION_BLOCK FB_MKS909 EXTENDS FB_GaugeBase

VAR_INPUT
	PG	: ST_VG;
END_VAR
VAR_OUTPUT
	{attribute 'pytmc' := '
    pv: 
	'}
	IG	: ST_VG;
END_VAR
VAR_IN_OUT
	
END_VAR
VAR
	rV : REAL;
	rMaxPressure	:	REAL := 5E-2; //Torr
	rMinPressure	:	REAL := 1E-10; //Torr
	timer:TON;
	(*Default set point 50 mT*)
	rVAC_SP: REAL := 9E-3; // as per manual
	iTermBits: UINT := 30518 ; // The terminal's maximum value in bits default el3174 as per vacuum architecture
	(*IO*)
	i_iPRESS_R AT%I* :INT; // input Pressure // Link to analog Input
	q_xHV_DIS AT %Q* : BOOL := True; // Active Low 
	
END_VAR

(* Standard MKS 9XX series conversion *)
(* works for 972 and 925 *)

//Default setpoint 50 mT
IF PG.rVAC_SP = 0 THEN
	PG.rVAC_SP := rVAC_SP;
END_IF
// check no div by zero
If (iTermBits=0) THEN iTermBits := 30518;END_IF
rV := 10*INT_TO_REAL(PG.i_iPRESS_R)/iTermBits;

(* Pressure OK check *)
// Gauge state
// Is the gauge plugged in, and within a reasonable range?
IF  (rV >= 0.1 and rV <=8.7) THEN // as per manual
	IG.rPRESS := LREAL_TO_REAL(EXPT(10, rV-10));
	IG.eState := Valid;
	IG.xPRESS_OK := TRUE; //Backwards compatibility
ELSIF rV > 8.7 AND rV < 10 THEN
	IG.rPRESS :=rMaxPressure;
	IG.xPRESS_OK := FALSE;
	IG.eState := Off;
ELSE 
	IG.xPRESS_OK := FALSE;
	IG.eState := GaugeDisconnected;
END_IF


IF (PG.rPRESS <= IG.rPRO_SP)  AND (PG.xPRESS_OK) THEN
		 PG.q_xHV_DIS := NOT IG.xHV_SW;
		 IG.xILKOk := TRUE;
	ELSIF NOT IG.q_xHV_DIS AND timer.Q THEN
		IF IG.rPRESS > (IG.rPRO_SP + IG.rHYS_PR) OR PG.rPRESS > (IG.rPRO_SP + IG.rHYS_PR) THEN
		IG.q_xHV_DIS := TRUE;
		IG.xHV_SW := FALSE;
		END_IF
	ELSE 
		IG.q_xHV_DIS := TRUE;
		IG.xHV_SW := FALSE;
		IG.xILKOk := FALSE;
 	END_IF
 

timer(IN:= NOT IG.q_xHV_DIS, PT:= T#2s);

(* Setpoint evaluation *)
IG.xAT_VAC := IG.xPRESS_OK AND (IG.rPRESS < IG.rVAC_SP);

(*Soft IO Mapping*)
ACT_IO();

(*Logger*)

THIS^.ACT_Logger();

ACTION ACT_IO:
(*soft link inputs*)
IG.i_iPRESS_R:=	i_iPRESS_R; 

(*soft link outputs*)
q_xHV_DIS := IG.q_xHV_DIS;
END_ACTION

ACTION ACT_Logger:
// ILK logger
IF NOT IG.xILKOk AND NOT IG.q_xHV_DIS THEN
 		fbLogger(sMsg:='Lost external interlock while gauge was on.', eSevr:=TcEventSeverity.Critical);  	
END_IF


// Log Action
tAction(CLK:=  IG.q_xHV_DIS);
IF tAction.Q THEN fbLogger(sMsg:='Ion gauge commanded to switch on', eSevr:=TcEventSeverity.Info); END_IF



//STATE Logger  
IF ePrevState <> IG.eState THEN
	  CASE IG.eState OF
		ValidHi:
		ValidLo:
		Valid:
			fbLogger(sMsg:='Gauge pressure valid.', eSevr:=TcEventSeverity.Info);
  		GaugeDisconnected:
			fbLogger(sMsg:='Gauge Disconnected.', eSevr:=TcEventSeverity.Critical);
		PressInvalid:
			fbLogger(sMsg:='Gauge pressure invalid.', eSevr:=TcEventSeverity.Warning);
		OoR:
			fbLogger(sMsg:='Gauge pressure out of range.', eSevr:=TcEventSeverity.Warning);
		Starting:
			fbLogger(sMsg:='Gauge starting.', eSevr:=TcEventSeverity.Info);
	  END_CASE
	  ePrevState := IG.eState;  
  END_IF
END_ACTION

METHOD M_AutoOn : BOOL
VAR_INPUT
END_VAR
this^.IG.q_xHV_DIS:= FALSE;
END_METHOD

METHOD M_SetBits : BOOL
VAR_INPUT
	TermBits : UINT; // The terminal's maximum value in bits
END_VAR
This^.iTermBits := TermBits;
END_METHOD

END_FUNCTION_BLOCK

// POUs/Functions/Pumps/functions/F_TurboExtILK_NO
(* This function Block interfaces with a NO turbo valve*)
(* Mainly used in the FEE HXR GATT*)
FUNCTION F_TurboExtILK_NO : BOOL
VAR_INPUT
	Turbo		:	ST_PTM;
	BackingGauge:	ST_VG;
	InletGauge	:	ST_VG;
	VentValve	:	ST_VCC_NO; //NO type turbo valve
	ScrollPump	:	ST_RoughPump;
END_VAR

VAR
END_VAR

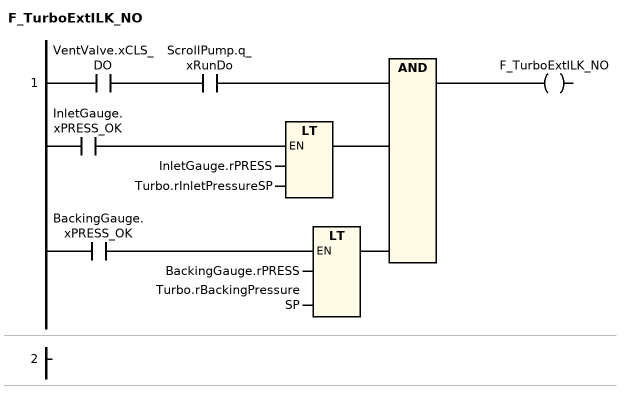
// NETWORK 1
F_TurboExtILK_NO := (VentValve.xCLS_DO AND ScrollPump.q_xRunDo) AND (InletGauge.xPRESS_OK AND InletGauge.rPRESS < Turbo.rInletPressureSP) AND (BackingGauge.xPRESS_OK AND BackingGauge.rPRESS < Turbo.rBackingPressureSP);

// NETWORK 2

END_FUNCTION

// POUs/Functions/Pumps/functions/F_TurboExtILK_NO_1
(* This function Block interfaces with a NO turbo valve*)
(* Mainly used in the FEE HXR GATT*)
FUNCTION F_TurboExtILK_NO_1 : BOOL
VAR_INPUT
	Turbo		:	ST_PTM;
	BackingGauge:	ST_VG;
	InletGauge	:	ST_VG;
	VentValve	:	ST_VCC_NO; //NO type turbo valve
	ScrollPump	:	ST_RoughPump;
END_VAR

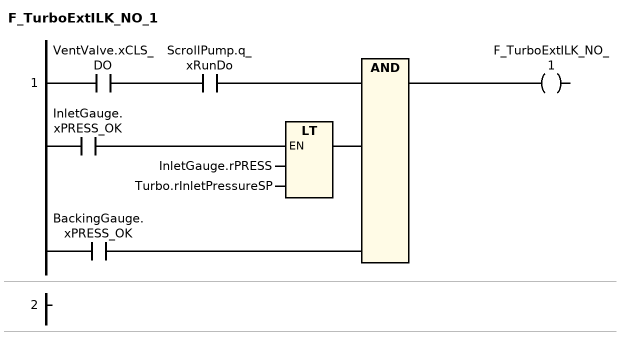
// NETWORK 1
F_TurboExtILK_NO_1 := (VentValve.xCLS_DO AND ScrollPump.q_xRunDo) AND (InletGauge.xPRESS_OK AND InletGauge.rPRESS < Turbo.rInletPressureSP) AND BackingGauge.xPRESS_OK;

// NETWORK 2

END_FUNCTION

// POUs/Functions/Pumps/functions/F_TurboExtILKLogic

(* This function evaluates the Turbo ILK logic*)
(* The Turbo shall not Run if the vent valve is open*)
(* The function also switches off the Turbo if the Inlet pressure or the backing Pressure*)
(* are higher than the configured set point*)
FUNCTION F_TurboExtILKLogic : BOOL
VAR_INPUT
	Turbo		:	ST_PTM;
	BackingGauge:	ST_VG;
	InletGauge	:	ST_VG;
	VentValve	:	ST_VVC;
	ScrollPump	:	ST_RoughPump;
END_VAR

VAR
END_VAR

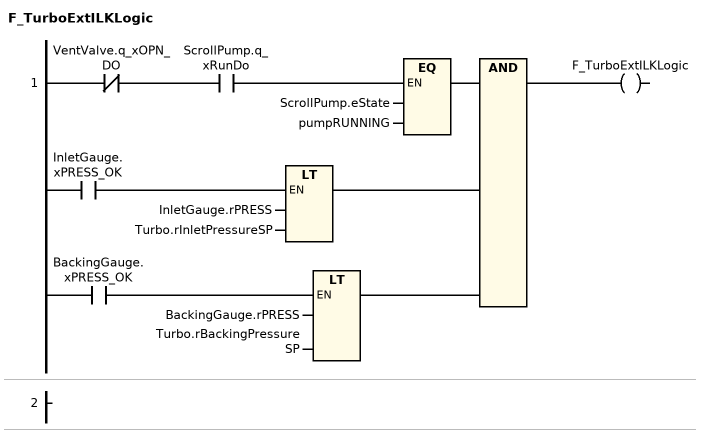
// NETWORK 1
F_TurboExtILKLogic := (NOT VentValve.q_xOPN_DO AND ScrollPump.q_xRunDo AND ScrollPump.eState = pumpRUNNING) AND (InletGauge.xPRESS_OK AND InletGauge.rPRESS < Turbo.rInletPressureSP) AND (BackingGauge.xPRESS_OK AND BackingGauge.rPRESS < Turbo.rBackingPressureSP);

// NETWORK 2

END_FUNCTION

// POUs/Functions/Pumps/functions/F_TurboExtILKLogic_2

(* This function evaluates the Turbo ILK logic*)
(* The function switches off the Turbo if the Inlet pressure or the backing Pressure*)
(* are higher than the configured set point*)
FUNCTION F_TurboExtILKLogic_2 : BOOL
VAR_INPUT
	Turbo		:	ST_PTM;
	BackingGauge:	ST_VG;
	InletGauge	:	ST_VG;
	ScrollPump	:	ST_RoughPump;
END_VAR
VAR
END_VAR

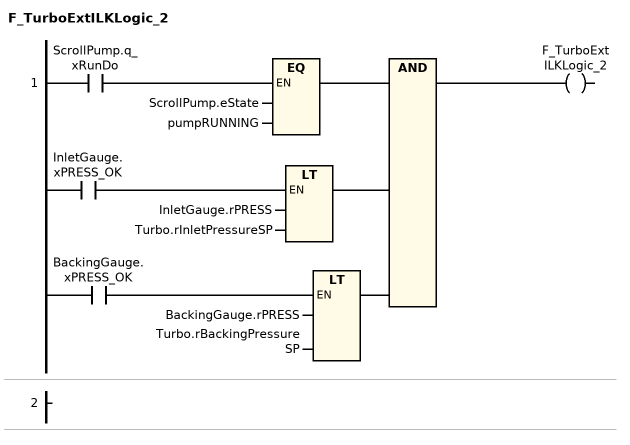
// NETWORK 1
F_TurboExtILKLogic_2 := (ScrollPump.q_xRunDo AND ScrollPump.eState = pumpRUNNING) AND (InletGauge.xPRESS_OK AND InletGauge.rPRESS < Turbo.rInletPressureSP) AND (BackingGauge.xPRESS_OK AND BackingGauge.rPRESS < Turbo.rBackingPressureSP);

// NETWORK 2

END_FUNCTION

// POUs/Functions/Pumps/functions/FB_TurboExtLogic
(*deprecated*)
FUNCTION_BLOCK FB_TurboExtLogic
VAR_IN_OUT
	Turbo		:	ST_AgilentPTM;
END_VAR
VAR_INPUT
	BackingGauge:	ST_VG;
	InletGauge	:	ST_VG;
	VentValve	:	ST_VCC_NO;
	ScrollPump	:	ST_RoughPump;
END_VAR
VAR_OUTPUT
END_VAR
VAR
END_VAR

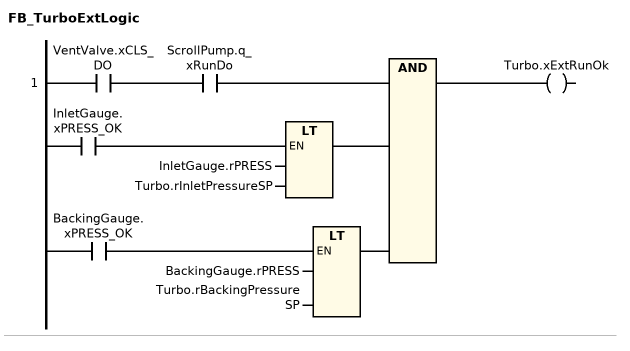
// NETWORK 1
Turbo.xExtRunOk := (VentValve.xCLS_DO AND ScrollPump.q_xRunDo) AND (InletGauge.xPRESS_OK AND InletGauge.rPRESS < Turbo.rInletPressureSP) AND (BackingGauge.xPRESS_OK AND BackingGauge.rPRESS < Turbo.rBackingPressureSP);

END_FUNCTION_BLOCK

// POUs/Functions/Pumps/Interfaces/FB_PIP_Interface_In
(* This function block is created for interface devices between different PLC*)
(* Not all the Variables in the original structure is required, just few signals *)
(* They have to be linked to the custom created variables on the EL6692/5 primary side*)
FUNCTION_BLOCK FB_PIP_Interface_In
VAR_INPUT
END_VAR
VAR_OUTPUT
	VG : ST_VG;
END_VAR
VAR
	i_rPRESS AT%I*: REAL;  //This is the human-readable pressure
	i_xAT_VAC AT%I*: BOOL;
	i_xPRESS_OK AT%I*: BOOL;
	i_xIs_Connected AT%I*: BOOL;
END_VAR

(* This function block is created for interface devices between different PLC*)
(* Not all the Variables in the original structure is required, just few signals *)
(* They have to be linked to the custom created variables on the EL6692/5 primary side*)

VG.rPRESS := i_rPRESS;
VG.xAT_VAC := i_xAT_VAC;
VG.xPRESS_OK := i_xPRESS_OK;


IF NOT(i_xIs_Connected) THEN
	i_xPRESS_OK := FALSE;
END_IF

END_FUNCTION_BLOCK

// POUs/Functions/Pumps/Interfaces/FB_PIP_Interface_Out
(* This function block is created for interface devices between different PLC*)
(* Not all the Variables in the original structure is required, just few signals *)
(* They have to be linked to the custom created variables on the EL6692/5 primary side*)
FUNCTION_BLOCK FB_PIP_Interface_Out
VAR_INPUT
	VG : ST_VG;
END_VAR
VAR_OUTPUT
END_VAR
VAR
	i_rPRESS AT%Q*: REAL; 
	i_xAT_VAC AT%Q*: BOOL;
	i_xPRESS_OK AT%Q*: BOOL;
END_VAR

(* This function block is created for interface devices between different PLC*)
(* Not all the Variables in the original structure is required, just few signals *)
(* They have to be linked to the custom created variables on the EL6692/5 primary side*)

i_rPRESS:=VG.rPRESS;
i_xAT_VAC:= VG.xAT_VAC;
i_xPRESS_OK:=VG.xPRESS_OK;

END_FUNCTION_BLOCK

// POUs/Functions/Pumps/Interfaces/FB_TPIP_ADS
(* This function block is created for interface devices between different PLC*)
(* Not all the Variables in the original structure is required, just few signals *)
(* The variable values are read via ADS using the symbol name*)
FUNCTION_BLOCK FB_TPIP_ADS Extends FB_ADS
VAR_INPUT
	sNetId : String; //NetID of the Destination PLC controller
	nPort : uint; // port number
	sVarName : string;// the variable name of the declared pip/pin function block.
	iWatchdog:UDINT;//The watchdog variable name written to by the remote plc
END_VAR
VAR_OUTPUT
	{attribute 'pytmc' := 'pv:'}
	IG : ST_VG;
	bError: BOOL;
END_VAR
VAR
	fb_CheckWatchdog: FB_CheckWatchdog;
	fb_Read_VG: FB_ReadAdsSymByName;
	ftReset: F_TRIG;
	xFirstPass: BOOL:= true;
	
END_VAR


ftReset(CLK:= fb_Read_VG.bBusy OR xFirstPass);
xFirstPass := false;
(*calling ADS read function*)
	
fb_Read_VG(
	bRead:=ftReset.Q , 
	sNetId:= sNetId, 
	nPort:= nPort, 
	sVarName:= CONCAT(sVarName,'.q_IG'), 
	nDestAddr:= ADR(IG), 
	nLen:= SIZEOF(IG), 
	tTimeout:= , 
	eComMode:=eAdsComModeFastCom , 
	bBusy=> , 
	bError=> , 
	nErrorId=> );	
	

(*Error*)
fb_CheckWatchdog(
	bEnable:= TRUE, 
	tWatchdogTime:= T#900ms, 
	nCnt:= iWatchdog , 
	bWatchdog=> , 
	nLastCnt=> );

bError:= fb_Read_VG.bError OR fb_CheckWatchdog.bWatchdog;
tErrorPresent(CLK:=bError);

IF (fb_Read_VG.bError OR fb_CheckWatchdog.bWatchdog) THEN
IG.xPRESS_OK := FALSE;
END_IF;

(*Logger*)
ACT_Logger();

ACTION ACT_Logger:
IF tErrorPresent.Q THEN
 IF(fb_Read_VG.bError) THEN fbLogger(sMsg:='ADS Read Error', eSevr:=TcEventSeverity.Critical); END_IF;
 IF(fb_CheckWatchdog.bWatchdog) THEN fbLogger(sMsg:='ADS Watchdog Error', eSevr:=TcEventSeverity.Critical); END_IF;
END_IF
END_ACTION

END_FUNCTION_BLOCK

// POUs/Functions/Pumps/FB_EbaraDryPump
(*This function block does basic controls for the Ebara EV-S Dry pump. Starts booster pump when appropriate. Turns off pump
in the event of errors/ warnings. Provides interlocking interface.*)
FUNCTION_BLOCK FB_EbaraDryPump EXTENDS FB_Pump
VAR_INPUT
	i_stBPGauge	:	ST_VG; //booster pump interlock gauge
	i_xVlvOpn	:	BOOL; //valve(s) to main system load are open
	i_xExtIlkOK	:	BOOL;
	
END_VAR
VAR_OUTPUT
	{attribute 'pytmc' := '
    pv: 
	'}
	stPump	:	ST_EbaraDryPump; //Ebara dry pump structure
END_VAR
VAR_IN_OUT
	
END_VAR
VAR
	(*IO*)
	q_xMPStart	AT%Q*:	BOOL; //Main Pump start
	q_xBPStart	AT%Q*:	BOOL; // Booster Pump start (this can be started by the pump automatically)
	//Readbacks
	i_xMPStatus	AT%I*:	BOOL; //MP status
	i_xBPStatus	AT%I*:	BOOL; //BP status
	i_xWarning	AT%I*:	BOOL; //Warning status
	i_xAlarmOK	AT%I*:	BOOL; //Alarm, maps to error
	i_xRemote	AT%I*:	BOOL; //Remote control status
END_VAR

(* Ebara Dry Pump Control Routine
A. Wallace
2016-4-29
Applicable to:
EV-S20
EV-S50
EV-S100
EV-S200

Does basic controls for the pump. Starts booster pump when appropriate. Turns off pump
in the event of errors/ warnings. Provides interlocking interface.

Main Pump Operational Note:
Ebara recommends that the pump be exposed to the full system load after the main pump is running.

Booster Pump Operational Note:
The booster pump can either be started automatically by the pump itself (probably based on a timer?)
or it can be started by the PLC. The pressure setpoint is by default 30T. It may be wise to make
sure the pump was exposed to the full system load before starting the booster.

*)

//Mapping
ACT_IO();
stPump.xExtIlk := NOT i_xExtIlkOK;

//Interlock and error/warning
stPump.xIlkOK :=  NOT stPump.xExtIlk AND NOT (stpump.xErr);// OR stpump.xWrn);

//Start/ Stop the pump
IF stpump.xIlkOK THEN
	stpump.q_xMPStart := stpump.pv_xRunSW;
ELSE
	stpump.q_xMPStart := stpump.pv_xRunSW := FALSE;
END_IF

//Booster pump
stpump.xBPIlk := i_xVlvOpn AND stpump.i_xMPStatus AND (i_stBPGauge.rPRESS < stpump.rBPIlkSP) AND i_stbpgauge.xPRESS_OK;
stpump.tonBP(IN:=stpump.xBPIlk);
stpump.q_xBPStart := stpump.tonBP.Q;

(*State evaluation*)
IF stPump.i_xAlarm THEN
	stpump.eState := pumpFAULT;
ELSIF NOT stpump.q_xMPStart AND stPump.i_xAlarm THEN
		stpump.eState := pumpSTOPPED;	
ELSIF stpump.q_xMPStart AND NOT stPump.i_xMPStatus THEN
		stpump.eState := pumpSTARTING;	
ELSIF stPump.i_xMPStatus OR stPump.i_xBPStatus THEN
		stpump.eState := pumpRUNNING;
ELSIF NOT stPump.i_xMPStatus AND NOT stPump.i_xBPStatus THEN
		stpump.eState := pumpSTOPPED;
ELSE
	stpump.eState := pumpFAULT;
END_IF


//Mapping
ACT_IO();
// Log States and triggers
ACT_Logger();

ACTION ACT_IO:
(*Outputs*)
q_xMPStart	:= stPump.q_xMPStart;
q_xBPStart	:= stPump.q_xBPStart;
stPump.q_xRunDo := stPump.q_xMPStart;
(*Inputs*)
stPump.i_xMPStatus:=	i_xMPStatus;
stPump.i_xBPStatus:=	i_xBPStatus;
stPump.i_xWarning:= NOT i_xWarning;
// These are normally closed inputs
stPump.xWrn := NOT i_xWarning;
stPump.i_xAlarm:=	NOT(i_xAlarmOK);
StPump.xErr := NOT(i_xAlarmOK);
stPump.i_xRemote:= i_xRemote;
END_ACTION

ACTION ACT_Logger:
// ILK logger
IF NOT i_xExtIlkOK AND ePrevState = pumpRUNNING THEN
 		fbLogger(sMsg:='Lost external interlock while pump was running.', eSevr:=TcEventSeverity.Critical);  	
END_IF
//STATE Logger  

IF ePrevState <> stpump.eState THEN
	  CASE stpump.eState OF
		pumpFAULT:
			fbLogger(sMsg:='Pump Fault.', eSevr:=TcEventSeverity.Critical);
  		pumpSTOPPED:
			fbLogger(sMsg:='Pump stopped.', eSevr:=TcEventSeverity.Critical);
		pumpSTARTING:
			fbLogger(sMsg:='Pump starting.', eSevr:=TcEventSeverity.Info);
		pumpRUNNING:
			fbLogger(sMsg:='Pump running.', eSevr:=TcEventSeverity.Info);
	  END_CASE
	  ePrevState := stpump.eState;  
  END_IF
  

// Log Action
tAction(CLK:=  stPump.q_xRunDo);
IF tAction.Q THEN fbLogger(sMsg:='Pump commanded to start', eSevr:=TcEventSeverity.Info); END_IF


// Log FAULT
tFault(CLK:= NOT stPump.i_xAlarm);
IF tFault.Q THEN fbLogger(sMsg:='Pump Lost Alarm OK bit', eSevr:=TcEventSeverity.Critical); END_IF
END_ACTION

END_FUNCTION_BLOCK

// POUs/Functions/Pumps/FB_Pump
FUNCTION_BLOCK FB_Pump
VAR_INPUT
END_VAR
VAR_OUTPUT
END_VAR
VAR
	
 // For logging
    fbLogger : FB_LogMessage := (eSubsystem:=E_SubSystem.VACUUM);
    ePrevState : E_PumpState;
    tErrorPresent : R_TRIG;
    tAction : R_TRIG; // Primary action of this device (OPN_DO, PUMP_RUN, etc.)	
	tFault : F_TRIG;
	tILK: TON;
END_VAR

ACTION ACT_Logger:

END_ACTION

END_FUNCTION_BLOCK

// POUs/Functions/Pumps/FB_EbaraEVA
(*This function block does basic controls for the Ebara EV-A  pump. Turns off pump
in the event of errors/ warnings. Provides interlocking interface.*)
FUNCTION_BLOCK FB_EbaraEVA EXTENDS FB_Pump
VAR_INPUT
	i_xExtIlkOK	:	BOOL;
END_VAR
VAR_OUTPUT
	{attribute 'pytmc' := '
    pv: 
	'}
	stPump	:	ST_EbaraEVA; //Ebara dry pump structure 
END_VAR
VAR
  // For logging
  (*  fbLogger : FB_LogMessage := (eSubsystem:=E_SubSystem.VACUUM);
    ePrevState : E_PumpState;
    tErrorPresent : R_TRIG;
    tAction : R_TRIG; // Primary action of this device (OPN_DO, PUMP_RUN, etc.)	
	tFault : F_TRIG;*)

(*IO*)
	q_xRunDo AT%Q* : BOOL; // Output signal
	q_xRemote At%Q* :BOOL;// Remote/Local Control
	q_xResetAlarm At%Q* :BOOL;// Remote/Local Control
	i_xAlarmOK AT%I* :BOOL; // Normally closed Alarm bit
	i_xIsRun   AT%I*:BOOL; // Input status
END_VAR

(*MG 2019*)
stPump.xIlkOK := i_xExtIlkOK AND stPump.i_xAlarmOK ;
// Enable the remote signal when the interlock evaluation is ok
//stPump.q_xRemote := stPump.xIlkOK;

IF stPump.xIlkOK THEN
	stPump.q_xRunDO := stPump.pv_xRunSW;
ELSE
		stPump.PV_xRunSW := FALSE;
        stPump.q_xRunDO := FALSE;
END_IF

(*State evaluation*)
IF NOT(stPump.i_xAlarmOK ) THEN
	 ePrevState := stpump.eState;
	stpump.eState := pumpFAULT;
ELSIF NOT stpump.q_xRunDo AND stPump.i_xAlarmOK THEN
		stpump.eState := pumpSTOPPED;	
ELSIF NOT stpump.q_xRunDo AND NOT stPump.i_xIsRun THEN
		stpump.eState := pumpSTARTING;	
ELSIF stPump.i_xIsRun THEN
		stpump.eState := pumpRUNNING;
ELSE
	stpump.eState := pumpFAULT;
END_IF


//Soft IO Mapping
ACT_IO();

// Log States and triggers
ACT_Logger();

ACTION ACT_IO:
stPump.i_xAlarmOK:=	i_xAlarmOK;
stPump.xErr:=	NOT(i_xAlarmOK);
stPump.i_xIsRun := i_xIsRun;
(*outputs*)
q_xRunDo:=stPump.q_xRunDo;
q_xRemote:= stPump.q_xRemote;
END_ACTION

ACTION ACT_Logger:
// ILK logger
IF NOT i_xExtIlkOK AND ePrevState = pumpRUNNING THEN
 		fbLogger(sMsg:='Lost external interlock while pump was running.', eSevr:=TcEventSeverity.Critical);  	
END_IF

//STATE Logger  
IF ePrevState <> stpump.eState THEN
	  CASE stpump.eState OF
		pumpFAULT:
			fbLogger(sMsg:='Pump Fault.', eSevr:=TcEventSeverity.Critical);
  		pumpSTOPPED:
			fbLogger(sMsg:='Pump stopped.', eSevr:=TcEventSeverity.Critical);
		pumpSTARTING:
			fbLogger(sMsg:='Pump starting.', eSevr:=TcEventSeverity.Info);
		pumpRUNNING:
			fbLogger(sMsg:='Pump running.', eSevr:=TcEventSeverity.Info);
	  END_CASE
	  ePrevState := stpump.eState;  
  END_IF
  
// Log Action
tAction(CLK:=  stPump.q_xRunDo);
IF tAction.Q THEN fbLogger(sMsg:='Pump commanded to start', eSevr:=TcEventSeverity.Info); END_IF


// Log FAULT
tFault(CLK:= stPump.i_xAlarmOK);
IF tFault.Q THEN fbLogger(sMsg:='Pump Lost Alarm OK bit', eSevr:=TcEventSeverity.Critical); END_IF
END_ACTION

END_FUNCTION_BLOCK

// POUs/Functions/Pumps/FB_KashiyamaPump
(* This function block does basic controls FOR the Kashiyama pump. Turns off pump
in the event of errors/ warnings. Provides interlocking interface.*)
FUNCTION_BLOCK FB_KashiyamaPump
VAR_IN_OUT

END_VAR
VAR_INPUT
	
END_VAR
VAR_OUTPUT
	{attribute 'pytmc' := 'pv:'}
	q_stPump : ST_KashiyamaDryPump;
END_VAR
VAR
	TONtmr : TON;
	resetTmr : TON;
	
	(* Output *)	
	q_xRunDO 	AT%Q*:	BOOL;
	q_xResetDo	AT%Q*: 	BOOL;
	q_xLspdDo	AT%Q*: 	BOOL;
	
(* Input *)
	i_xLocal	AT%I*:	BOOL;
	i_xAlarm	AT%I*:	BOOL;
	i_xWarning	AT%I*:	BOOL;
	i_xIsRun	AT%I*:	BOOL;
END_VAR


//Kashiyama Dry pump outputs at high level indicate no warning, no alarm and remotely
q_stPump.xIlkOK := q_stPump.i_xLocal AND q_stPump.i_xWarningOK AND q_stPump.i_xAlarmOK;

IF q_stPump.xIlkOK THEN
	q_stPump.q_xRunDO := q_stPump.pv_xRunSW;
	ELSE
		q_stPump.PV_xRunSW := FALSE;
        q_stPump.q_xRunDO := FALSE;	
END_IF
 
q_stPump.xLspd_IlkENA := q_stPump.q_xRunDO;

IF q_stPump.xLspd_IlkENA THEN
	q_stPump.q_xLspdDo := q_stPump.xLspdSW;
	ELSE
		q_stPump.xLspdSW := FALSE;
        q_stPump.q_xLspdDo := FALSE;	
END_IF

//resetTmr (In := iq_stPump.xResetSW, PT := T#2S);
//IF resetTmr.Q THEN
//	iq_stPump.xResetSW := FALSE;
//END_IF

q_stPump.q_xResetDo := NOT q_stPump.i_xIsRun AND q_stPump.xResetSW;

//countdown Timer
TONtmr (IN := q_stPump.i_xIsRun, PT := T#20S);
q_stPump.RdyTmr := TO_REAL(TONtmr.PT) - TO_REAL(TONtmr.ET);

(*State evaluation*)
IF NOT q_stPump.i_xAlarmOK THEN
	q_stPump.eState := pumpFAULT;
ELSIF NOT q_stPump.q_xRunDo AND q_stPump.i_xAlarmOK THEN
		q_stPump.eState := pumpSTOPPED;	
ELSIF NOT q_stPump.q_xRunDo AND NOT q_stPump.i_xIsRun THEN
		q_stPump.eState := pumpSTARTING;	
ELSIF q_stPump.i_xIsRun THEN
		q_stPump.eState := pumpRUNNING;
ELSE
	q_stPump.eState := pumpFAULT;
END_IF

//Mapping
ACT_IO();

ACTION ACT_IO:
(* Output *)	
	q_xRunDO 	:= q_stPump.q_xRunDO;
	q_xResetDo := q_stPump.q_xResetDo;;
	q_xLspdDo := q_stPump.q_xLspdDo;;
	
(* Input *)
	q_stPump.i_xLocal := i_xLocal;
	q_stPump.i_xAlarmOK :=	i_xAlarm;
	q_stPump.i_xWarningOK :=	i_xWarning;
	q_stPump.i_xIsRun :=	i_xIsRun;
END_ACTION

METHOD PUBLIC M_Run : BOOL
VAR_INPUT
	run:bool; // set to true to run, false to stop;
END_VAR

this^.q_stPump.pv_xRunSW := run;
END_METHOD

END_FUNCTION_BLOCK

// POUs/Functions/Pumps/FB_PIP_Gamma
(* This function block does basic controls FOR the ION pump connected to a Gamma QPCe controller.
 Provides interlocking interface. Enable HV only when interlock gauge press is less than 1.0E-4 Torr *)
{attribute 'reflection'} 
FUNCTION_BLOCK FB_PIP_Gamma Extends FB_Pump
VAR_INPUT
	i_stGauge	:	ST_VG; //Ion or Pirani gauge for pump interlock
    i_xOverrideMode : BOOL; (*To be linked to global override bit. This Overrides Vacuum interlock logic*) 
END_VAR
VAR_OUTPUT
	{attribute 'pytmc' := '
    pv: 
	'}
	stPump	:	ST_PIP; //Gamma Ion pump structure
	q_IG	:	ST_VG; //When ion pump is used as a measuring device for interlocking gate valves
END_VAR
VAR_IN_OUT
END_VAR
VAR
 rPRESS : REAL;
 
 rV : REAL;
 timer:TON; 
 rHVEna_SP : REAL :=1E-4; // Default protection setpoint as per the gamma QPCe manual
 (* IO Controls *)
 q_xHVEna_DO AT %Q*: BOOL;	// Enable High Voltage when TRUE
 i_iPRESS  AT %I*: INT;  //
 i_xSP_DI  AT %I* : BOOL; // NO contact //function of relay set on the QPC to HV output state

// For logging
tTimeOutAction : F_TRIG;
tOverrideActivated : R_TRIG;

tPumpStartTimeout : TON := (PT:=T#10s); // Timeout pump start if pressure < 1E-11 for more than 10s.
MinPressure : REAL:= 1E-11; // Minimum readback pressure, pump must register pressure above this to be considered running
 
//Overrides
	tonOvrd	:	TON;
	tonDelOK : TON;
	rtOK	:	R_TRIG;
	tOvrd	:	TIME := T#10s;
	
	{attribute 'instance-path'}
	{attribute 'noinit'}
	sPath: STRING;
END_VAR

(* Does Gamma Ion pump HV interlock. Enable HV only when interlock gauge press is less than 1.0E-4 Torr *)

(*Ensures the set point is not higher than 1.0E-4*)
IF (stPump.rHVEna_SP > rHVEna_SP) THEN
	stPump.rHVEna_SP := rHVEna_SP;
END_IF

(* Interlock *)
//stPump.xHV_ExtIlk  := i_stGauge.xPRESS_OK AND (i_stGauge.rPRESS <= stPump.rHVEna_SP);//AND NOT tPumpStartTimeout.Q); //ADP

(* Enable HV *)
IF i_stGauge.rPRESS <= stPump.rHVEna_SP AND i_stGauge.xPRESS_OK THEN
	IF (stPump.xAutoOn) AND NOT (stPump.q_xHVEna_DO) THEN  stPump.q_xHVEna_DO := TRUE;
	ELSE stPump.q_xHVEna_DO := stPump.xHVEna_SW OR ((tonOvrd.Q AND i_xOverrideMode));  
	END_IF
	stPump.xILKOk:= TRUE;
ELSIF stPump.q_xHVEna_DO (*AND timer.Q*) THEN 
	IF q_IG.rPRESS > (stPump.rHVEna_SP + stPump.rHYS_PR) THEN // Ion pumps when running switches off based on their own pressure readings
		stPump.q_xHVEna_DO := FALSE;
		stPump.xHVEna_SW := FALSE;
		stPump.xILKOk := FALSE;
	ELSE
		stPump.q_xHVEna_DO := stPump.xHVEna_SW OR ((tonOvrd.Q AND i_xOverrideMode)); 
	END_IF
ELSIF (tonOvrd.Q AND i_xOverrideMode) THEN
	stPump.q_xHVEna_DO := TRUE;
ELSE
	stPump.q_xHVEna_DO  := FALSE;
	stPump.xHVEna_SW := FALSE;
	stPump.xILKOk := FALSE;
END_IF


//stPump.q_xHVEna_DO := stPump.xHVEna_SW AND stPump.xHV_ExtIlk;
//stPump.xHVEna_SW := stPump.q_xHVEna_DO;

timer(IN:= NOT stPump.q_xHVEna_DO, PT:= T#1s);

// TAW Experimental ion pump timeout
tPumpStartTimeout(IN:=(NOT stPump.i_xHV_DI AND stPump.q_xHVEna_DO));
tTimeOutAction(CLK:=tPumpStartTimeout.Q);
IF tTimeOutAction.Q THEN  fbLogger(sMsg:='Pump time out.', eSevr:=TcEventSeverity.Critical); END_IF



(*Pump STATE*)
IF tPumpStartTimeout.Q THEN //Pump timeout
	stPump.eState := pumpFAULT;
ELSIF stPump.q_xHVEna_DO AND NOT stPump.i_xHV_DI THEN
	stPump.eState := pumpSTARTING;
ELSIF NOT stPump.q_xHVEna_DO AND NOT stPump.i_xHV_DI THEN
	stPump.eState := pumpSTOPPED;
ELSIF stPump.q_xHVEna_DO AND stPump.i_xHV_DI THEN
	stPump.eState := pumpRUNNING;
ELSIF NOT stPump.q_xHVEna_DO AND stPump.i_xHV_DI THEN
	stPump.eState := pumpSTOPPING;
ELSE 
	stPump.eState := pumpFAULT;
END_IF



(*Update output gauge values*)
ACT_SetGauge();
(*Soft IO Mapping*)
IO();
ACT_IlkOverride();
// Log States and triggers
ACT_Logger();

ACTION ACT_IlkOverride:
(* Override logic *)
(* Goal: give ability to override, but do so in a way that people won't forget it.
Solution: Override only after ten seconds of override, protect against blips,
when the Pump permission goes true for more than ten seconds consistently, remove override
*)

tonDelOK(IN:=stPump.xILKOk, PT:=T#10S);
rtOK(CLK:=tonDelOK.Q);
IF rtOK.Q AND stPump.pv_xOvrdStart THEN 
	stPump.pv_xOvrdStart :=FALSE; 
	if (stPump.eState = pumpRUNNING) AND (i_xOverrideMode) THEN stPump.xHVEna_SW:= TRUE; END_IF
    //Log
    fbLogger(sMsg:='Override expired', eSevr:=TcEventSeverity.Warning);
END_IF
// Release the Force DO bit when the system override is false
IF NOT(i_xOverrideMode) THEN stPump.pv_xOvrdStart :=FALSE; END_IF
//Override timer
tonOvrd(IN:= stPump.pv_xOvrdStart, PT:=tOvrd);
END_ACTION

ACTION ACT_Logger:
// ILK logger

IF NOT (stPump.xILKOk) AND ((ePrevState = pumpRUNNING) OR (ePrevState = pumpSTARTING)) AND NOT tonOvrd.Q THEN 
	fbLogger(sMsg:='Pump turned off due to loss of interlock.', eSevr:=TcEventSeverity.Critical); 
END_IF

//STATE Logger  
IF ePrevState <> stPump.eState THEN
	  CASE stPump.eState OF
		pumpFAULT:
			fbLogger(sMsg:='Pump Fault.', eSevr:=TcEventSeverity.Critical);
  		pumpSTOPPED:
			fbLogger(sMsg:='Pump stopped.', eSevr:=TcEventSeverity.Critical);
		pumpSTARTING:
			fbLogger(sMsg:='Pump starting.', eSevr:=TcEventSeverity.Info);
		pumpRUNNING:
			fbLogger(sMsg:='Pump running.', eSevr:=TcEventSeverity.Info);
		pumpSTOPPING:
			fbLogger(sMsg:='Pump stopping.', eSevr:=TcEventSeverity.Info);
	  END_CASE
	  ePrevState := stPump.eState;  
  END_IF

  
  // Log Action
tAction(CLK:=  stPump.q_xHVEna_DO);
IF tAction.Q THEN fbLogger(sMsg:='Pump commanded to start', eSevr:=TcEventSeverity.Info); END_IF
// Log override mode enabled
tOverrideActivated(CLK:= (tonOvrd.Q AND i_xOverrideMode));
IF tOverrideActivated.Q THEN fbLogger(sMsg:='Pump override mode activated', eSevr:=TcEventSeverity.Warning); END_IF


// Log FAULT
tFault(CLK:=  NOT tPumpStartTimeout.Q);
IF tFault.Q THEN fbLogger(sMsg:='Pump Fault', eSevr:=TcEventSeverity.Critical); END_IF
END_ACTION

ACTION ACT_SetGauge:
(*MG*)
(* convert the analog input into readable pressure*)
(* use logarithmic Pressure calculation, Output= Normal and Offset = 0*)
rV := 10*INT_TO_REAL(i_iPress)/32767;
//Manual Page 9

if (stPump.bOutputInverted) THEN
	rPRESS := LREAL_TO_REAL(EXPT(10,(rV-stPump.iOffset)*-1));
ELSE 
	rPRESS := LREAL_TO_REAL(EXPT(10,(rV-stPump.iOffset)));
END_IF
IF (stPump.q_xHVEna_DO) THEN
	q_IG.rPRESS := rPRESS;
	stPump.rPRESS := rPRESS;
END_IF


IF (stPump.i_xHV_DI) AND (q_IG.rPRESS < q_IG.rVAC_SP) THEN //ADP// AND (q_IG.rPRESS<>0) AND stPump.q_xHVEna_DO) THEN 
	q_IG.xPRESS_OK := TRUE;
	ELSE
	q_IG.xPRESS_OK := FALSE;
END_IF

q_IG.sPath := This^.stPump.sPath;
END_ACTION

ACTION IO:
stPump.sIlkDeviceName := This^.i_stGauge.sPath;
stPump.xError := (stPump.eState = pumpFAULT);
stPump.xOverrideMode := i_xOverrideMode; 
(*inputs*)
stPump.i_iPRESS:=	i_iPRESS;  
stPump.i_xHV_DI:=	i_xSP_DI;
(*output*)
q_xHVEna_DO:=  stPump.q_xHVEna_DO; //According to Manual pin should be grounded to activate function

 This^.stPump.sPath:= sPath;
END_ACTION

METHOD M_AutoOn : BOOL
VAR_INPUT
END_VAR
this^.stPump.xAutoOn:= TRUE; // Pump is set to auto start when the pressure is low enough
END_METHOD


METHOD PUBLIC M_Run : BOOL
VAR_INPUT
	run:bool; // set to true to run, false to stop;
END_VAR

this^.stPump.xHVEna_SW := run;
END_METHOD

END_FUNCTION_BLOCK

// POUs/Functions/Pumps/FB_PTM_Agilent
(* This function block does basic controls FOR the Agilent TV Turbo pump. Turns off pump
in the event of errors/ warnings. Provides interlocking interface.*)
FUNCTION_BLOCK FB_PTM_Agilent EXTENDS FB_Pump
VAR_IN_OUT
	
END_VAR
VAR_INPUT
	i_xExtILKOk : BOOL; // Connect to external interlock logic(e.g TURBO_ILK Function), TRUE if not used.
	i_stGauge	:	ST_VG; //Pirani backing gauge for pump interlock 
	i_rMaxBackingPressure : REAL;
END_VAR
VAR_OUTPUT
	{attribute 'pytmc' :=' pv:'}
	iq_stPtm	:	ST_AgilentPTM;	
	
END_VAR
VAR
	{attribute 'instance-path'}
	{attribute 'noinit'}
	sPath: STRING;
	//xRunOk	:	BOOL;
	nMaxR1Fault: INT :=5;
	nR1Fault : INT;
	tFaultWindowDuration : TIME := T#300S;
	tR1FaultDuration : TIME := T#120S;
	tTimeOutDuration: TIME:= T#10M;
	tFaultWindowElapsed: TON;
	tR1Fault : TON;
	tStartTimeOut : TON;
	tR1TimeOut: TON;
	step : INT :=0;
	nErrorCode: INT :=0;
	xBackingPressureOK: BOOL;
	iMaxSpeed : INT:=963;
	
	rPowerScale: REAL:=10;//W
	rCurrentScale: REAL:=1;//A
	
	(*I/Os*)
	i_xSTART 	AT%I*:	BOOL;
	i_xR1	AT%I*	:  BOOL;
	i_xR2	AT%I*	:  BOOL;
	i_xLSpd	AT%I*:  BOOL;
	i_iTempMon AT%I*: INT;
	i_iPowerMon AT%I*: INT;
	i_iCurrentMon AT%I*: INT;
	i_iRawSpeed AT %I* : INT; 
	i_xFault AT%I*	:	BOOL;
	q_RunDO AT%Q*	:	BOOL;
	q_xLSpd	AT%Q*	:  BOOL;
    
    
    // For logging
  //  Msg : FB_FormatString;
   // fbJson : FB_JsonSaxWriter;
   tOverrideActivated : R_TRIG;
	
	iTermBits: UINT := 32767 ; // The terminal's maximum value in bits
END_VAR

(* Basic Agilent Turbo Controls *)
(* M. Ghaly, 2018-9-26 *)

(*connect External interlock to structure variable*)
//iq_stPtm.xExtRunOk := i_xExtILKOk;

(* state machine *)
CASE (step) OF
(*Pump Stopped State*)
	0: // Pump Stopped State
		iq_stPtm.xRunSW:=FALSE;
		//Reset Output signals;
		iq_stPtm.q_RunDO:=FALSE;
		iq_stPtm.q_xSS := FALSE;
		iq_stPtm.q_xLSpd:= FALSE;
		//Reset timer
		tFaultWindowElapsed.IN := FALSE;
		nR1Fault := 0;
		iq_stPtm.eState := pumpSTOPPED;
		step :=10;
        
(*Idle State waiting to start*)	
	10: // Idle State, waiting for the xRunSwitch
		IF iq_stPtm.xExtRunOk  AND iq_stPTM.xRunSW THEN
			iq_stPtm.q_RunDO := iq_stPTM.xRunSW; //
			step:=20;
		END_IF
(*Pump Starting State*)	
	20: // Pump is starting
		nErrorCode:=0;
		iq_stPtm.q_RunDO := iq_stPTM.xRunSW; // done in previous state
		IF (*(NOT iq_stPtm.i_xR1) AND*)iq_stPtm.i_xSTART  THEN
		iq_stPtm.eState := pumpSTARTING;
		step:= 40;
		ELSIF tStartTimeOut.Q THEN
			step:=90; // or fault state
			nErrorCode:=950;
		END_IF
		// should check R1 ?? check Fault condition?
        
		
	40: // Pump is starting
		iq_stPtm.eState := pumpSTARTING;
		IF   NOT iq_stPtm.i_xR1 AND NOT iq_stPtm.i_xSTART  THEN
			step := 0 ;
		ELSIF NOT iq_stPtm.i_xR1 AND iq_stPtm.i_xSTART  THEN
			step :=40;
		ELSIF iq_stPtm.i_xR1 AND NOT iq_stPtm.i_xSTART THEN
			step:= 50;
		END_IF
		IF tR1TimeOut.Q THEN
			step:= 90;
			iq_stPtm.xPumpFaultLock := TRUE;
			nErrorCode:= 930; // R1 Signal at Start time out.
           // fbLogger(sMsg:='Timeout: Pump could not achieve running speed.', eSevr:=TcEventSeverity.Warning);
		END_IF
		
	50: // Pump is Running (Normal Operation) ( R1 is True and STARTing is FALSE)
		iq_stPtm.eState := pumpRUNNING;
		IF NOT iq_stPtm.i_xR1 THEN
			nR1Fault:= nR1Fault+1 ; 
			tFaultWindowElapsed.IN := TRUE; ///
			//tR1Fault.IN := TRUE;
			step :=60;
		END_IF
        
        //Log new state
        IF ePrevState <> iq_stPtm.eState THEN
            //fbLogger(sMsg:='Pump at speed.', eSevr:=TcEventSeverity.Verbose);
            ePrevState := iq_stPtm.eState;
		END_IF
	
	60: // Pump is Running (Not Nomral Operation) (R1 is False, pump not @ speed )
		IF ((nR1Fault = nMaxR1Fault) AND NOT tFaultWindowElapsed.Q) OR (tR1Fault.Q) THEN // number of fault occured during the same time window
			step:= 90;
			tR1Fault.IN := FALSE;
			tFaultWindowElapsed.IN := FALSE;
			iq_stPtm.xPumpFaultLock := TRUE;
			nErrorCode:= 920; // R1 Signal Lost multiple times.
            //fbLogger(sMsg:='Running signal Lost multiple times.', eSevr:=TcEventSeverity.Warning);
		ELSIF tFaultWindowElapsed.Q  THEN
			tFaultWindowElapsed.IN := FALSE;
			nR1Fault := 0;
		ELSIF iq_stPtm.i_xR1 THEN
			tR1Fault.IN := FALSE;
			step:=50;
		END_IF
	
	90: // Pump Fault STATE 
		iq_stPtm.xRunSW:=FALSE;
		iq_stPtm.q_RunDO:=FALSE;
		iq_stPtm.q_xSS := FALSE;
		iq_stPtm.q_xLSpd:= FALSE;
		iq_stPtm.eState := pumpFAULT;
		step := 95;
	
	95:	
		IF (NOT iq_stPtm.xPumpFaultLock) OR iq_stPtm.xRunSW THEN 
			step:=0;
		END_IF
END_CASE

(* Interrupts *)
(* FAULT signal*)
IF (iq_stPtm.i_xFault) AND (step < 90 ) THEN 
	iq_stPtm.eState := pumpFAULT; // no need taken care of in the state
	iq_stPtm.xPumpFaultLock := TRUE;
	nErrorCode := 900; // Pump Controller FAULT
	step:=90; 
END_IF


(*Pump Lock Reset bit*)
IF (iq_stPtm.xResetSW ) THEN
	iq_stPtm.xResetSW := FALSE;
	iq_stPtm.xPumpFaultLock := FALSE;
END_IF

(*Check backing gauge pressure*)
//xBackingPressureOK := i_stGauge.xPRESS_OK AND ( i_stGauge.rPRESS < iq_stPtm.rBackingPressureSP);

(* Interlock Sum *)
iq_stPtm.xExtRunOk := i_xExtILKOk AND NOT iq_stPtm.i_xFault AND NOT iq_stPtm.xPumpFaultLock AND NOT(tILK.Q);

IF NOT iq_stPtm.xExtRunOk AND (NOT (step >= 90)) THEN
	step:=0; 
END_IF

(*Stop By the Operator and not due to fault *)
IF (NOT iq_stPtm.xRunSW) AND (NOT (step >= 90)) AND (NOT (step = 10)) THEN
	step := 0;
END_IF

// Log faults Moved to ACT_Logger
(*tErrorPresent(CLK:=iq_stPtm.xPumpFaultLock);
IF tErrorPresent.Q THEN
    fbJson.StartObject();
    fbJson.AddKey('vacuum_typecode');
    fbJson.AddUdint(nErrorCode);
    fbJson.EndObject();
    fbLogger.sJson := fbJson.GetDocument();
    fbLogger(sMsg:='Turbo control fault', eSevr:=TcEventSeverity.Warning);
    fbJson.ResetDocument();
END_IF
*)

(* Timers *)
tFaultWindowElapsed(PT:=tFaultWindowDuration);
tR1Fault(IN:= (step = 60), PT:=tR1FaultDuration);
tStartTimeOut(IN := (step=20), PT:=tTimeOutDuration);
tR1TimeOut(IN := (step=40), PT:=tTimeOutDuration);
(* IO Mapping*)
IO();
(*Assign Error Message*)
iq_stPtm.sError := ErrorMessage(nErrorCode, iq_stPtm.eState);
// Log States and triggers
ACT_Logger();
(*Validate Backing Pressure set point doesn't exceed the Maximum backingPressure*)
iq_stPtm.rBackingPressureSP := BackingPressureSetPoint(iq_stPtm.rBackingPressureSP,i_rMaxBackingPressure);
ACT_Interlock();

ACTION ACT_Interlock:
This^.tILK(IN:= (i_stGauge.rPRESS>=iq_stPtm.rBackingPressureSP), PT:=T#5S, Q=> );
END_ACTION

ACTION ACT_Logger:
//STATE Logger  
// ILK logger
IF NOT i_xExtIlkOK AND ePrevState = pumpRUNNING THEN
 		fbLogger(sMsg:='Lost external interlock while pump was running.', eSevr:=TcEventSeverity.Critical);  	
END_IF


IF ePrevState <> iq_stPTM.eState THEN
	  CASE iq_stPTM.eState OF
		pumpFAULT:
			fbLogger(sMsg:='Pump Fault.', eSevr:=TcEventSeverity.Critical);
  		pumpSTOPPED:
			fbLogger(sMsg:='Pump stopped.', eSevr:=TcEventSeverity.Critical);
		pumpSTARTING:
			fbLogger(sMsg:='Pump starting.', eSevr:=TcEventSeverity.Info);
		pumpRUNNING:
			fbLogger(sMsg:='Pump running.', eSevr:=TcEventSeverity.Info);
	  END_CASE
	  ePrevState := iq_stPTM.eState;  
  END_IF
  
// Log Action
tAction(CLK:=  iq_stPTM.q_RunDO);
IF tAction.Q THEN fbLogger(sMsg:='Pump commanded to start', eSevr:=TcEventSeverity.Info); END_IF


// Log FAULT
tFault(CLK:= iq_stPTM.i_xFault OR iq_stPtm.xPumpFaultLock);
IF tFault.Q THEN fbLogger(sMsg:=iq_stPtm.sError, eSevr:=TcEventSeverity.Critical); END_IF
END_ACTION

METHOD BackingPressureSetPoint : REAL
VAR_INPUT
	i_SetPoint : REAL;
	rMaxBackingPressure: REAL;
END_VAR
BackingPressureSetPoint := Min(i_SetPoint , rMaxBackingPressure);
END_METHOD

METHOD PUBLIC ErrorMessage : STRING
VAR_INPUT
	nErrorCode : INT;
	eState: E_PumpState;
END_VAR
IF (eState = pumpFAULT ) THEN
	CASE nErrorCode OF
		950:
			ErrorMessage := 'Pump Starting Fault';
		930: 
			ErrorMessage := 'Pump could not achieve running speed';
	
		920:
			ErrorMessage := 'Running at speed signal lost multiple times';

		900:
			ErrorMessage := 'Pump Controller Fault';	
	END_CASE
	
END_IF
END_METHOD

ACTION IO:
(*inputs*)
iq_stPtm.i_xSTART:=	i_xSTART;
iq_stPtm.i_xR1:=	i_xR1;
iq_stPtm.i_xR2:=	i_xR2;
iq_stPtm.i_xLSpd:=	i_xLSpd;
iq_stPtm.i_xFault:=	i_xFault;
(* Real-value calculation *)
If (iTermBits=0) THEN iTermBits := 32767;END_IF
iq_stPtm.i_rCurrentMon := (10*INT_TO_REAL(i_iCurrentMon)/iTermBits)*rCurrentScale; 
iq_stPtm.i_rTempMon := 10*INT_TO_REAL(i_iTempMon)/iTermBits; 
iq_stPtm.i_rPowerMon := (10*INT_TO_REAL(i_iPowerMon)/iTermBits)*rPowerScale; 
iq_stPtm.i_diCurSpd := 10*LREAL_TO_DINT(INT_TO_REAL(i_iRawSpeed)/iTermBits);


(*outputs*)
q_RunDO := iq_stPtm.q_RunDO;
q_xLSpd := iq_stPtm.q_xLSpd;
END_ACTION

METHOD PUBLIC M_Run : BOOL
VAR_INPUT
	run:bool; // set to true to run, false to stop;
END_VAR

this^.iq_stPtm.xRunSW := run;
END_METHOD

METHOD M_SetBits : BOOL
VAR_INPUT
	TermBits : UINT; // The terminal's maximum value in bits
END_VAR
This^.iTermBits := TermBits;
END_METHOD

METHOD M_SetCurrentScale : BOOL
VAR_INPUT
	Scale:REAL;//In Amps
END_VAR
This^.rCurrentScale := Scale;
END_METHOD

METHOD M_SetMaxSpeed : BOOL
VAR_INPUT
	iMaxSpeed: INT; //963Hz for 3.1,300HT and 1010Hz for 401 and 1350 for 81
END_VAR
this^.iMaxSpeed := iMaxSpeed;
END_METHOD

METHOD M_SetPowerScale : BOOL
VAR_INPUT
	Scale:REAL;//In Watt
END_VAR
This^.rPowerScale := Scale;
END_METHOD

METHOD PUBLIC M_TurboIsOn : BOOL
VAR_INPUT
END_VAR
M_TurboIsOn := (This^.iq_stPtm.eState =  E_PumpState.pumpSTARTING ) OR (This^.iq_stPtm.eState =  E_PumpState.pumpRUNNING );
END_METHOD

END_FUNCTION_BLOCK

// POUs/Functions/Pumps/FB_PTM_Ebara_010M
(* This function block does basic controls FOR the Ebara Turbo pump connected to the ETC010M Controller.
 Turns off pump in the event of errors/ warnings. Provides interlocking interface.*)
 {attribute 'no_check'}
FUNCTION_BLOCK FB_PTM_Ebara_010M EXTENDS FB_Pump
VAR_IN_OUT
	
END_VAR
VAR_INPUT
	i_xExtILKOk : BOOL; // Turbo ILK bit , set to True if not used
	//i_iRawSpeed: INT; //Should come from PLC Soft IO.
	i_rMaxBackingPressure : REAL := 3;
	i_iMinSpeed : DINT := 100; //Hz check pump manual for setting P43
	i_iMaxSpeed : DINT := 560; //Hz check pump manual for setting P43
END_VAR
VAR_OUTPUT
	{attribute 'pytmc' := '
    pv: 
	'}
	iq_stPTM : ST_EbaraPTM;
END_VAR
VAR
	i_iADCBits : UINT := 15;
	RTRIG_INLK: R_TRIG;
	TOF_RESET: TON :=(PT:=T#1S);
	TOF_SetSpeed: TON :=(PT:=T#1S);
	
	(*IO*)
	(*inputs*)
	i_xDecel AT %I* : BOOL; //Link to brake input
	i_xAccel AT %I* : BOOL;
	i_xRotate AT %I* : BOOL;
	i_xNCFault AT %I* : BOOL;// 
	i_xAtSpd AT %I* : BOOL;
	i_iRawSpeed AT %I* : INT; // Link to Analog input
	i_iTempMon AT %I* : INT; // Link to Analog input -- input Voltage according to the pump temprature 0->5V 0->100C
	i_iCurrentMon AT %I* : INT; //Link to Analog -- input Voltage to the output current of motor 0->5V 0->10A
	
	(*output*)
	q_xStart AT %Q* : BOOL; // link to output
	q_xStop AT %Q* : BOOL; //Link to output
	q_xReset AT %Q* : BOOL;
	q_xProtection AT %Q* : BOOL;
	q_xSetSpeed AT %Q* : BOOL;
	q_iSpeedSet AT %Q* :INT;	//Link to analog Output

END_VAR

(* Ebara ETC control FB
Scott Stubbs & Alex W.
Modified Nov 2018 by M. Ghaly
*)
(* The pump runs when the RunDO is set to true. The RunDO sets the outputs Start and Stop to true when it 
is true, and false otherwise. Per the manual, when START bit is closed the pump will accelerate, and when the STOP
bit is Opened, the pump will decelerate with the brake and stop *)

(* Simple protection reset *)
iq_stPtm.xExtRunOk:= i_xExtILKOk AND NOT iq_stPTM.i_xFault;
iq_stPTM.q_xProtection:= TRUE;//iq_stPTM.xExtRunOk;
(*soft IO mapping*)
ACT_IO();

(* Basic pump supervisory section *)
	(* If override mode, ignore everything else *)
IF iq_stPTM.i_xOverride THEN
	IF iq_stPTM.xRunSW THEN
		iq_stPTM.q_RunDO:=TRUE;
	ELSE
		iq_stPTM.q_RunDO:=FALSE;
	END_IF
	//Handle faults 
ELSIF iq_stPTM.i_xFault OR ( NOT iq_stPTM.xExtRunOk) THEN
	iq_stPTM.q_RunDO:=FALSE;
	iq_stPTM.xRunSW:=FALSE;
	//And one for when we need to start the pump normally. Only allows pump to be started if ILK ok.
ELSIF iq_stPTM.xRunSW AND iq_stPTM.xExtRunOk THEN
	iq_stPTM.q_RunDO:=TRUE;
END_IF
//One section for when pump is told to stop
IF NOT iq_stPTM.xRunSW THEN
		iq_stPTM.q_RunDO:=FALSE;
		//IF (NOT iq_stPTM.i_xFault)(* AND (NOT iq_stPTM.i_xALARM) *)THEN iq_stPTM.eState := pumpSTOPPED; END_IF;
END_IF 

//Set the Start and Stop outputs to Run do . check manual alternate START/STOP
iq_stPTM.q_xStart := iq_stPTM.q_RunDO;
iq_stPTM.q_xStop := iq_stPTM.q_RunDO; 



 (* to reset the Input speed OK bit *)
 TOF_SetSpeed (IN:= iq_stPTM.iq_xSpeedSet, Q => );
 IF  (TOF_SetSpeed.Q) THEN iq_stPTM.iq_xSpeedSet:= FALSE; 
 END_IF
 (* to reset the Reset Bit *)
 IF (iq_stPTM.xResetSW ) THEN  iq_stPTM.q_xReset := TRUE; 
 END_IF
 TOF_RESET (IN:= iq_stPTM.q_xReset, Q => );
 IF TOF_RESET.Q THEN 
	iq_stPTM.q_xReset:= FALSE;
	iq_stPTM.xResetSW := FALSE; 
 END_IF
 (*When the Protection signal is lost, Error bit doesn't show, but the controller still needs to be reset*)
RTRIG_INLK(CLK:= iq_stPTM.q_xProtection );
 IF (RTRIG_INLK.Q) AND (iq_stPTM.i_xNCFault) THEN
	 iq_stPTM.q_xReset := TRUE; 
 END_IF
 

 
(*Validate Backing Pressure set point doesn't exceed the Maximum backingPressure*)
iq_stPtm.rBackingPressureSP := BackingPressureSetPoint(iq_stPtm.rBackingPressureSP,i_rMaxBackingPressure);


 (*Pump STATE*)
IF iq_stPtm.i_xFault THEN 
	iq_stPtm.eState := pumpFAULT;
ELSIF iq_stPTM.i_xDecel AND NOT iq_stPtm.q_RunDO THEN
	iq_stPtm.eState := pumpSTOPPING;
ELSIF NOT iq_stPtm.q_RunDO AND NOT iq_stPTM.i_xFault THEN
	iq_stPtm.eState := pumpSTOPPED;
ELSIF NOT iq_stPtm.i_xAtSpd  AND iq_stPtm.q_RunDO AND iq_stPTM.i_xAccel THEN
	iq_stPtm.eState := pumpSTARTING;
ELSIF iq_stPtm.i_xAtSpd AND iq_stPtm.q_RunDO THEN
	iq_stPtm.eState := pumpRUNNING;
ELSE 
	iq_stPtm.eState := pumpFAULT;
END_IF

(*soft IO mapping*)
ACT_IO();
// Log States and triggers
ACT_Logger();

ACTION ACT_IO:
(*soft io mapping*)
(*inputs*)
	iq_stPTM.i_xDecel := i_xDecel ;
	iq_stPTM.i_xAccel :=	i_xAccel ;
	iq_stPTM.i_xRotate :=	i_xRotate;
	iq_stPTM.i_xFault := NOT iq_stPTM.i_xNCFault; 	//Normally closed fault handling
	iq_stPTM.i_xNCFault :=	i_xNCFault ;
	iq_stPTM.i_xALARM:= NOT i_xNCFault;
	iq_stPTM.i_xAtSpd := i_xAtSpd;
	iq_stPTM.i_rTempMon := (100*(INT_TO_REAL(i_iTempMon)/16383));// Manual page 28(DC 0 to 5V -> 0 to 100 DegC)
	iq_stPTM.i_rCurrentMon := (10*(INT_TO_REAL(i_iCurrentMon)/16383));// Manual page 28 (DC 0 to 5V -> 0 to 10 A)
	iq_stPTM.i_diCurSpd := LREAL_TO_DINT(560*LREAL_TO_DINT(i_iRawSpeed)/16383);//(560*(INT_TO_REAL(i_iRawSpeed)/16383));// Manual page 28 (DC 0 to 5V -> 100 to 560Hz Rated Rotational Speed )
(*outputs*)
	q_xStart:= iq_stPTM.q_xStart;
	q_xStop := iq_stPTM.q_xStop;
	q_xReset := iq_stPTM.q_xReset;
	q_xProtection := iq_stPTM.q_xProtection;
	q_xSetSpeed := iq_stPTM.iq_xSpeedSet;


(*Validate Set Speed within range *) 
IF iq_stPTM.q_iSpeedSet  >= i_iMinSpeed AND iq_stPTM.q_iSpeedSet  <=i_iMaxSpeed THEN 
	q_iSpeedSet  := LIMIT(0, DINT_TO_INT((iq_stPTM.q_iSpeedSet - i_iMinSpeed) / i_iMaxSpeed *16383/5),16383); //Max 5V
END_IF
END_ACTION

ACTION ACT_Logger:

IF NOT i_xExtIlkOK AND (ePrevState = pumpRUNNING OR ePrevState = pumpSTARTING) THEN
 		fbLogger(sMsg:='Pump turned off due to loss of interlock.', eSevr:=TcEventSeverity.Critical);  	
END_IF
// Log Action
tAction(CLK:=  iq_stPTM.q_RunDO);
IF tAction.Q THEN fbLogger(sMsg:='Pump commanded to start', eSevr:=TcEventSeverity.Info); END_IF



//STATE Logger  
IF ePrevState <> iq_stPTM.eState THEN
	  CASE iq_stPTM.eState OF
		pumpFAULT:
			fbLogger(sMsg:='Pump Fault.', eSevr:=TcEventSeverity.Critical);
  		pumpSTOPPED:
			fbLogger(sMsg:='Pump stopped.', eSevr:=TcEventSeverity.Critical);
		pumpSTARTING:
			fbLogger(sMsg:='Pump starting.', eSevr:=TcEventSeverity.Info);
		pumpRUNNING:
			fbLogger(sMsg:='Pump running.', eSevr:=TcEventSeverity.Info);
		pumpSTOPPING:
			fbLogger(sMsg:='Pump decelerating.', eSevr:=TcEventSeverity.Info);
	  END_CASE
	  ePrevState := iq_stPTM.eState;  
  END_IF
  

// Log FAULT
tFault(CLK:= iq_stPTM.i_xNCFault);
IF tFault.Q THEN fbLogger(sMsg:='Pump Lost Alarm OK bit', eSevr:=TcEventSeverity.Critical); END_IF
END_ACTION

METHOD PUBLIC BackingPressureSetPoint : REAL
VAR_INPUT
	i_SetPoint : REAL;
	rMaxBackingPressure: REAL;
END_VAR
BackingPressureSetPoint := Min(i_SetPoint , rMaxBackingPressure);
END_METHOD

METHOD PUBLIC M_Run : BOOL
VAR_INPUT
	run:bool; // set to true to run, false to stop;
END_VAR

this^.iq_stPtm.xRunSW := run;
END_METHOD

END_FUNCTION_BLOCK

// POUs/Functions/Pumps/FB_PTM_Ebara_011M
(* This function block does basic controls FOR the Ebara Turbo pump connected to the ETC011M Controller.
 Turns off pump in the event of errors/ warnings. Provides interlocking interface.*)
{attribute 'no_check'}
FUNCTION_BLOCK FB_PTM_Ebara_011M EXTENDS FB_Pump
VAR_IN_OUT
END_VAR
VAR_INPUT
	i_rMaxBackingPressure : REAL := 3;
	i_iMinSpeed : DINT := 100; //check pump manual for setting
	i_iMaxSpeed : DINT := 560; // check pump manual for setting
	i_xExtILKOk : BOOL; // Connect to external interlock logic, TRUE if not used.
END_VAR
VAR_OUTPUT
	{attribute 'pytmc' := '
    pv: 
	'}
	iq_stPTM : ST_EbaraPTM;
END_VAR
VAR
	TOF_SetSpeed: TON := (PT:=T#1S);
	TOF_RESET: TON :=(PT:=T#1S);
	i_iADCBits : UINT := 12;
	(*IO*)
	(*inputs*)
	i_xDecel AT %I* : BOOL; //Link to brake input
	i_xAccel AT %I* : BOOL;
	i_xRotate AT %I* : BOOL;
	i_xFaultNC AT %I* : BOOL;// remove?
	i_xAtSpd AT %I* : BOOL;
	i_iRawSpeed AT %I* : INT; // Link to Analog input
	
	(*output*)
	q_xStart AT %Q* : BOOL; // link to output
	q_xStop AT %Q* : BOOL; //Link to output
	q_xReset AT %Q* : BOOL;
	q_xProtection AT %Q* : BOOL;
	q_xSetSpeed AT %Q* : BOOL;
	q_iSpeedSet AT %Q* :INT;	//Link to analog Output
	
	
END_VAR

(* Ebara ETC control FB
Scott Stubbs & Alex W.
Modified Nov 2018 by M. Ghaly
*)

(* Switch processing *)
//TOF_START.IN := iq_stPTM.i_xStart;
//TOF_START();
//TOF_STOP.IN  := iq_stPTM.i_xStop;
//TOF_STOP();
//TOF_RESET.IN := iq_stPTM.i_xReset;
//TOF_RESET();

(* Simple protection reset *)
iq_stPtm.xExtRunOk:= i_xExtILKOk;
iq_stPTM.q_xProtection := TRUE;//iq_stPTM.xExtRunOk;

(*soft IO mapping*)
ACT_IO();

(* Basic pump supervisory section *)
	(* If override mode, ignore everything else *)
IF iq_stPTM.i_xOverride THEN
	IF iq_stPTM.xRunSW THEN
		iq_stPTM.q_RunDO:=TRUE;
	ELSE
		iq_stPTM.q_RunDO:=FALSE;
	END_IF
	//Handle faults - the way the Ebara cable is done, xFault is normally closed
ELSIF iq_stPTM.i_xFault OR (iq_stPTM.q_RunDO AND NOT iq_stPTM.xExtRunOk) THEN
	iq_stPTM.q_RunDO:=FALSE;
	//iq_stPTM.q_xProtection:=FALSE;
	iq_stPTM.xRunSW:=FALSE;
	//And one for when we need to start the pump normally. Only allows pump to be started if ILK ok.
ELSIF iq_stPTM.xRunSW AND iq_stPTM.xExtRunOk THEN
	iq_stPTM.q_RunDO:=TRUE;
END_IF
//One section for when pump is told to stop
IF NOT iq_stPTM.xRunSW THEN
		iq_stPTM.q_RunDO:=FALSE;
		IF (NOT iq_stPTM.i_xFault) AND (NOT iq_stPTM.i_xALARM) THEN iq_stPTM.eState := pumpSTOPPED; END_IF;
END_IF 

//Set the Start and Stop outputs to Run do . check manual.
iq_stPTM.q_xStart := iq_stPTM.q_xStop := iq_stPTM.q_RunDO;

(* to reset the Input speed OK bit *)
 TOF_SetSpeed (IN:= iq_stPTM.iq_xSpeedSet, Q => );
 IF TOF_SetSpeed.Q THEN iq_stPTM.iq_xSpeedSet:= FALSE; 
 END_IF
 (* to reset the Reset Bit *)
 IF (iq_stPTM.xResetSW ) THEN  iq_stPTM.q_xReset := TRUE; 
 END_IF
 TOF_RESET (IN:= iq_stPTM.q_xReset, Q => );
 IF TOF_RESET.Q THEN 
	iq_stPTM.q_xReset:= FALSE;
	iq_stPTM.xResetSW := FALSE; 
 END_IF
 
 
 (*Pump STATE*)
IF iq_stPtm.i_xFault THEN 
	iq_stPtm.eState := pumpFAULT;
ELSIF iq_stPTM.i_xDecel AND NOT iq_stPtm.q_RunDO THEN
	iq_stPtm.eState := pumpSTOPPING;
ELSIF NOT iq_stPtm.q_RunDO AND NOT iq_stPTM.i_xFault THEN
	iq_stPtm.eState := pumpSTOPPED;
ELSIF NOT iq_stPtm.i_xAtSpd  AND iq_stPtm.q_RunDO THEN
	iq_stPtm.eState := pumpSTARTING;
ELSIF iq_stPtm.i_xAtSpd AND iq_stPtm.q_RunDO THEN
	iq_stPtm.eState := pumpRUNNING;
ELSE 
	iq_stPtm.eState := pumpFAULT;
END_IF

(*Validate Backing Pressure set point doesn't exceed the Maximum backingPressure*)
iq_stPtm.rBackingPressureSP := BackingPressureSetPoint(iq_stPtm.rBackingPressureSP,i_rMaxBackingPressure);


(*soft IO mapping*)
ACT_IO();
// Log States and triggers
ACT_Logger();

ACTION ACT_IO:
(*soft io mapping*)
(*inputs*)
	iq_stPTM.i_xDecel := i_xDecel ;
	iq_stPTM.i_xAccel :=	i_xAccel ;
	iq_stPTM.i_xRotate :=	i_xRotate;
	iq_stPTM.i_xNCFault :=	i_xFaultNC ;
	iq_stPTM.i_xAtSpd := i_xAtSpd;
	//iq_stPTM.i_iRawSpeed :=	i_iRawSpeed;
//V (AI/32767*10) * (33600 {Max RPM} - 100) / 5
(*outputs*)
	q_xStart:= iq_stPTM.q_xStart;
	q_xStop := iq_stPTM.q_xStop;
	q_xReset := iq_stPTM.q_xReset;
	q_xProtection := iq_stPTM.q_xProtection;
	q_xSetSpeed := iq_stPTM.iq_xSpeedSet;
(*Validate Set Speed within range *) 
IF iq_stPTM.q_iSpeedSet  >= i_iMinSpeed AND iq_stPTM.q_iSpeedSet  <=i_iMaxSpeed THEN 
	q_iSpeedSet  := LIMIT(0, DINT_TO_INT((iq_stPTM.q_iSpeedSet - i_iMinSpeed) / i_iMaxSpeed *16383/5),16383); //Max output 5V
	//:= DINT_TO_INT((iq_stPTM.q_iSpeedSet-100) / 33600 *32767/2); //Max 5V
END_IF

(* Pump speed calculation *)
iq_stPTM.i_diCurSpd := LREAL_TO_DINT(560*LREAL_TO_DINT(i_iRawSpeed)/16383);//(560*(INT_TO_REAL(i_iRawSpeed)/16383));// Manual page 28 (DC 0 to 5V -> 100 to 560Hz Rated Rotational Speed )
(*IF i_iRawSpeed / (EXPT(2,i_iADCBits)-1) * 10 >= 0.2 THEN //Speed reading appears zero at ~0.16V
iq_stPTM.i_diCurSpd := LREAL_TO_DINT(560*LREAL_TO_DINT(i_iRawSpeed)/16383);
//iq_stPTM.i_diCurSpd := LREAL_TO_DINT(i_iRawSpeed/(EXPT(2,i_iADCBits)-1)*67000);
//V (AI/(2^{# ADC bits} -1 ) * 10[ADC 10V scaling]) * (33600 [Max RPM] - 100) / 5
ELSE
	iq_stPTM.i_diCurSpd := 0;
END_IF*)

//Normally closed fault handling
iq_stPTM.i_xFault := NOT iq_stPTM.i_xNCFault; //??
END_ACTION

ACTION ACT_Logger:
//STATE Logger  
IF NOT i_xExtIlkOK AND ePrevState = pumpRUNNING THEN
 		fbLogger(sMsg:='Lost external interlock while pump was running.', eSevr:=TcEventSeverity.Critical);  	
END_IF


IF ePrevState <> iq_stPTM.eState THEN
	  CASE iq_stPTM.eState OF
		pumpFAULT:
			fbLogger(sMsg:='Pump Fault.', eSevr:=TcEventSeverity.Critical);
  		pumpSTOPPED:
			fbLogger(sMsg:='Pump stopped.', eSevr:=TcEventSeverity.Critical);
		pumpSTARTING:
			fbLogger(sMsg:='Pump starting.', eSevr:=TcEventSeverity.Info);
		pumpRUNNING:
			fbLogger(sMsg:='Pump running.', eSevr:=TcEventSeverity.Info);
		pumpSTOPPING:
			fbLogger(sMsg:='Pump decelerating.', eSevr:=TcEventSeverity.Info);
	  END_CASE
	  ePrevState := iq_stPTM.eState;  
  END_IF
  
// ILK logger



// Log Action
tAction(CLK:=  iq_stPTM.q_RunDO);
IF tAction.Q THEN fbLogger(sMsg:='Pump commanded to start', eSevr:=TcEventSeverity.Info); END_IF


// Log FAULT
tFault(CLK:= iq_stPTM.i_xNCFault);
IF tFault.Q THEN fbLogger(sMsg:='Pump Lost Alarm OK bit', eSevr:=TcEventSeverity.Critical); END_IF
END_ACTION

METHOD PUBLIC BackingPressureSetPoint : REAL
VAR_INPUT
	i_SetPoint : REAL;
	rMaxBackingPressure: REAL;
END_VAR
BackingPressureSetPoint := Min(i_SetPoint , rMaxBackingPressure);
END_METHOD

METHOD PUBLIC M_Run : BOOL
VAR_INPUT
	run:bool; // set to true to run, false to stop;
END_VAR

this^.iq_stPtm.xRunSW := run;
END_METHOD

END_FUNCTION_BLOCK

// POUs/Functions/Pumps/FB_PTM_MagDriveDigital
(* This function block does basic controls FOR the Leybold connected to the MagDriveDigital Controller.
 Turns off pump in the event of errors/ warnings. Provides interlocking interface.*)
FUNCTION_BLOCK FB_PTM_MagDriveDigital EXTENDS FB_Pump
VAR_IN_OUT
	
END_VAR
VAR_INPUT
	
	i_xExtILKOk : BOOL; // Connect to external interlock logic, TRUE if not used.
END_VAR
VAR_OUTPUT
{attribute 'pytmc' := '
    pv: 
	'}
	iq_stPtm	:	ST_LeyboldPTM;
END_VAR
VAR
	xRunOk	:	BOOL;
	tofRemoteDelay	:	TOF;
	
	
	(*IO*)
	i_xAtSpd AT%I*: BOOL; // Normaml operation when true
	i_xFault AT%I*: BOOL; // Error NC
    i_xAccel AT%I*: BOOL;
 	i_xDecel AT%I*: BOOL;
 	i_xWarn AT%I*: BOOL;
	
	q_RunDO AT%Q*: BOOL; // Start/Stop
	q_xRemote AT%Q*: BOOL;
END_VAR

(* Basic MagDrive Digital Turbo Controls *)
(* A. Wallace, 2015-7-15 *)

tofRemoteDelay(IN:=iq_stPtm.q_RunDO, PT:=T#5S);

iq_stPtm.q_xRemote := tofRemoteDelay.Q;

(* Interlock Sum *)
iq_stPtm.xExtRunOk:= i_xExtILKOk;
xRunOk := iq_stPtm.xExtRunOk AND NOT iq_stPtm.i_xFault;

(* Basic pump supervisory section *)
IF xRunOk THEN
	iq_stPtm.q_RunDO := iq_stPTM.xRunSW;
ELSE
	iq_stPtm.xRunSW:=FALSE;
	iq_stPtm.q_RunDO:=FALSE;
END_IF

(*Pump STATE*)
IF iq_stPtm.i_xFault THEN 
	iq_stPtm.eState := pumpFAULT;
ELSIF iq_stPTM.i_xDecel AND NOT iq_stPtm.q_RunDO THEN
	iq_stPtm.eState := pumpSTOPPING;
ELSIF NOT iq_stPtm.q_RunDO AND NOT iq_stPTM.i_xFault THEN
	iq_stPtm.eState := pumpSTOPPED;
ELSIF NOT iq_stPtm.i_xAtSpd  AND iq_stPtm.q_RunDO AND iq_stPTM.i_xAccel THEN
	iq_stPtm.eState := pumpSTARTING;
ELSIF iq_stPtm.i_xAtSpd AND iq_stPtm.q_RunDO THEN
	iq_stPtm.eState := pumpRUNNING;
ELSE 
	iq_stPtm.eState := pumpFAULT;
END_IF


(*I/O soft mapping*)
ACT_IO();
// Log States and triggers
ACT_Logger();

ACTION ACT_IO:
(*Inputs*)
iq_stPtm.i_xAtSpd := i_xAtSpd;
iq_stPtm.i_xFault := NOT i_xFault;
iq_stPtm.i_xAccel := i_xAccel;
iq_stPtm.i_xDecel := i_xDecel;
iq_stPtm.i_xWarn := i_xWarn;

(*Outputs*)
q_RunDO := iq_stPtm.q_RunDO;
q_xRemote := iq_stPtm.q_xRemote; // remote out
END_ACTION

ACTION ACT_Logger:
//STATE Logger  
IF NOT i_xExtIlkOK AND ePrevState = pumpRUNNING THEN
 		fbLogger(sMsg:='Lost external interlock while pump was running.', eSevr:=TcEventSeverity.Critical);  	
END_IF


IF ePrevState <> iq_stPTM.eState THEN
	  CASE iq_stPTM.eState OF
		pumpFAULT:
			fbLogger(sMsg:='Pump Fault.', eSevr:=TcEventSeverity.Critical);
  		pumpSTOPPED:
			fbLogger(sMsg:='Pump stopped.', eSevr:=TcEventSeverity.Critical);
		pumpSTARTING:
			fbLogger(sMsg:='Pump starting.', eSevr:=TcEventSeverity.Info);
		pumpRUNNING:
			fbLogger(sMsg:='Pump running.', eSevr:=TcEventSeverity.Info);
	  END_CASE
	  ePrevState := iq_stPTM.eState;  
  END_IF
  
// ILK logger



// Log Action
tAction(CLK:=  iq_stPTM.q_RunDO);
IF tAction.Q THEN fbLogger(sMsg:='Pump commanded to start', eSevr:=TcEventSeverity.Info); END_IF


// Log FAULT
tFault(CLK:= NOT iq_stPTM.i_xFault);
IF tFault.Q THEN fbLogger(sMsg:='Pump Lost Alarm OK bit', eSevr:=TcEventSeverity.Critical); END_IF
END_ACTION

METHOD PUBLIC M_Run : BOOL
VAR_INPUT
	run:bool; // set to true to run, false to stop;
END_VAR

this^.iq_stPtm.xRunSW := run;
END_METHOD

END_FUNCTION_BLOCK

// POUs/Functions/Pumps/FB_PTM_Pfeiffer
(* This function block does basic controls FOR the Pfeiffer Turbo pump connected to the TM700 and TC400 Controllers.
 Turns off pump in the event of errors/ warnings. Provides interlocking interface.*)
FUNCTION_BLOCK FB_PTM_Pfeiffer EXTENDS FB_Pump
VAR_IN_OUT
	
END_VAR
VAR_INPUT
	i_xExtIlkOK : BOOL; // Connect to external interlock logic, TRUE if not used.
END_VAR
VAR_OUTPUT
	{attribute 'pytmc' := '
    pv: 
	'}
	iq_stPTM : ST_PfeifferPTM;
END_VAR
VAR
	TOF_RESET: TON :=(PT:=T#1S);
	(*IO*)
	i_xAtSpd AT%I*: BOOL; // Normaml operation when true
	i_xFaultNC AT%I*: BOOL; // Error
	i_xWarn AT%I*: BOOL;
 	i_xRemote AT%I*: BOOL;
	
	q_RunDO AT%Q*: BOOL; // Start/Stop for TC110 link this output to the Pumping station bit
	q_PumpingStation AT%Q*: BOOL; // Start/Stop interlock
	q_xRemote AT%Q*: BOOL;
	q_xReset AT%Q*: BOOL;
END_VAR

(* Basic pump supervisory section *)

q_xRemote := TRUE;
(* Interlock Sum *)
iq_stPtm.xExtRunOk:= i_xExtILKOk;
//For compatability with TC110
(*IF iq_stPTM.xExtRunOk THEN
	q_PumpingStation:= TRUE;
ELSE 
	q_PumpingStation:= FALSE;
END_IF*)

IF iq_stPTM.xExtRunOk AND NOT (iq_stPTM.i_xFault) (*OR iq_stPTM.i_xTempFault)*) THEN
	iq_stPTM.q_RunDO:=iq_stPTM.xRunSW;
	q_PumpingStation:=iq_stPTM.xRunSW;
ELSE
	iq_stPTM.xRunSW:=FALSE;
	iq_stPTM.q_RunDO:=FALSE;
	q_PumpingStation:=FALSE;
END_IF


(*Pump STATE*)
IF iq_stPtm.i_xFault THEN 
	iq_stPtm.eState := pumpFAULT;
ELSIF NOT iq_stPtm.q_RunDO AND NOT iq_stPTM.i_xFault THEN
	iq_stPtm.eState := pumpSTOPPED;
ELSIF NOT iq_stPtm.i_xAtSpd  AND iq_stPtm.q_RunDO THEN
	iq_stPtm.eState := pumpSTARTING;
ELSIF iq_stPtm.i_xAtSpd AND iq_stPtm.q_RunDO THEN
	iq_stPtm.eState := pumpRUNNING;
ELSE 
	iq_stPtm.eState := pumpFAULT;
END_IF

(*Error Reset*)
(* to reset the Reset Bit *)
 IF (iq_stPTM.xResetSW ) THEN  
	iq_stPTM.q_xReset := TRUE; 
	q_PumpingStation := TRUE;
 END_IF

 IF (iq_stPTM.xResetSW) AND (iq_stPTM.i_xFault)  THEN  
	q_PumpingStation := TRUE;
 END_IF
 TOF_RESET (IN:= iq_stPTM.q_xReset, Q => );
 IF TOF_RESET.Q THEN 
	iq_stPTM.q_xReset:= FALSE;
	iq_stPTM.xResetSW := FALSE; 
 END_IF

(*Soft IO Mapping*)
ACT_IO();
// Log States and triggers
ACT_Logger();

ACTION ACT_IO:
(*outputs*)
q_RunDO := iq_stPTM.q_RunDO;
q_xReset := iq_stPTM.q_xReset;
//q_xRemote := iq_stPTM.
//q_PumpingStation AT%Q*: BOOL; // Start/Stop
	
(*inputs*)
iq_stPTM.i_xAtSpd:= i_xAtSpd;
iq_stPTM.i_xFault:= NOT i_xFaultNC; 
iq_stPTM.i_xWarn:=  	i_xWarn ;
END_ACTION

ACTION ACT_Logger:
//STATE Logger  
IF NOT i_xExtIlkOK AND ePrevState = pumpRUNNING THEN
 		fbLogger(sMsg:='Lost external interlock while pump was running.', eSevr:=TcEventSeverity.Critical);  	
END_IF


IF ePrevState <> iq_stPTM.eState THEN
	  CASE iq_stPTM.eState OF
		pumpFAULT:
			fbLogger(sMsg:='Pump Fault.', eSevr:=TcEventSeverity.Critical);
  		pumpSTOPPED:
			fbLogger(sMsg:='Pump stopped.', eSevr:=TcEventSeverity.Critical);
		pumpSTARTING:
			fbLogger(sMsg:='Pump starting.', eSevr:=TcEventSeverity.Info);
		pumpRUNNING:
			fbLogger(sMsg:='Pump running.', eSevr:=TcEventSeverity.Info);
	  END_CASE
	  ePrevState := iq_stPTM.eState;  
  END_IF
  
// ILK logger



// Log Action
tAction(CLK:=  iq_stPTM.q_RunDO);
IF tAction.Q THEN fbLogger(sMsg:='Pump commanded to start', eSevr:=TcEventSeverity.Info); END_IF


// Log FAULT
tFault(CLK:= NOT iq_stPTM.i_xFault);
IF tFault.Q THEN fbLogger(sMsg:='Pump Lost Alarm OK bit', eSevr:=TcEventSeverity.Critical); END_IF
END_ACTION

METHOD PUBLIC M_Run : BOOL
VAR_INPUT
	run:bool; // set to true to run, false to stop;
END_VAR

this^.iq_stPtm.xRunSW := run;
END_METHOD

METHOD PUBLIC M_Serial_IO : BOOL
VAR_INPUT
	st_Pfeiffer_RBK: ST_PfeifferStatus;
END_VAR
VAR_IN_OUT
	st_Pfeiffer_CTRL: ST_PfeifferControl;
END_VAR
(* This function block is used to map the IO points from the pfeiffer structures
to the generic turbo structures *)
(*
if (bInit) Then
	bInit := False;
	st_Pfeiffer_CTRL.diSetRotationSpeed_309 := st_Pfeiffer_RBK.diActiveRotationSpeed_309;
END_IF*)

(* Controls *) (* Controls is via DIO*)
//st_Pfeiffer_CTRL.xPumpingStation_010 := iq_stPTM.q_RunDO;
//st_Pfeiffer_CTRL.xMotorPump_023 := 1; //Setting always true because parameter 10 alone can enable/disable the pump
//st_Pfeiffer_CTRL.uiPowerPct_708 := iq_stPTM.q_uiPowerPct;
//st_Pfeiffer_CTRL.xErrorAck_009 := iq_stPTM.xResetSW;



(* Readbacks *)
iq_stPTM.i_xAccel := st_Pfeiffer_RBK.xPumpAccelerating_307;
//iq_stPTM.i_xAtSpd := st_Pfeiffer_RBK.xRotationSpeedAttn_306; The Atspd is already linked via Digital I/Os
iq_stPTM.i_diCurSpd := st_Pfeiffer_RBK.diActiveRotationSpeed_309;
iq_stPTM.i_diPwr := st_Pfeiffer_RBK.diDrivePower_316;
iq_stPTM.i_diElecTemp := st_Pfeiffer_RBK.diTempElec_326;
iq_stPTM.i_diBtmTemp := st_Pfeiffer_RBK.diTempPmpBot_330;
iq_stPTM.i_diBrngTemp := st_Pfeiffer_RBK.diTempBearng_342;
iq_stPTM.i_diMtrTemp := st_Pfeiffer_RBK.diTempMotor_346;
iq_stPTM.i_uiPowerPctRbk := st_Pfeiffer_RBK.uiPowerPct_708;
iq_stPTM.i_rCurrentMon :=  st_Pfeiffer_RBK.lrDriveCurrent_310;
iq_stPTM.xCommTimeout	:=	st_Pfeiffer_RBK.xTimeout;
iq_stPTM.i_iErrorCode := st_Pfeiffer_RBK.iErrorCode_303;
iq_stPTM.i_iWarningCode := st_Pfeiffer_RBK.iWarningCode_303;

(* Check that error acknowledgment is processed *)
IF st_Pfeiffer_RBK.xErrorAcknowledged THEN
	st_Pfeiffer_RBK.xErrorAcknowledged := FALSE;
	st_Pfeiffer_CTRL.xErrorAck_009 := FALSE;
	iq_stPTM.xResetSW := FALSE;
END_IF

IF st_Pfeiffer_RBK.sErrorCode_303 = '' THEN
	;
ELSIF st_Pfeiffer_RBK.sErrorCode_303 <> '000000' THEN
iq_stPTM.i_xFault := TRUE;
ELSE
iq_stPTM.i_xFault := FALSE;
END_IF

iq_stPTM.i_dSetSpd := LIMIT (0, iq_stPTM.i_dSetSpd, 1500); // 1500 nominal frequency
IF ( iq_stPTM.i_dSetSpd <>0) THEN
	st_Pfeiffer_CTRL.iSetRotationSpeed_707 := DINT_TO_INT(iq_stPTM.i_dSetSpd * 100/1500);
	st_Pfeiffer_CTRL.iSetRotationSpeed_707 := LIMIT(20, st_Pfeiffer_CTRL.iSetRotationSpeed_707 ,100); // Manual Page 18
END_IF
END_METHOD

END_FUNCTION_BLOCK

// POUs/Functions/Pumps/FB_PTM_TurboDrive
(* This Function block provides basic turbo control for Leybold Turbo Drive 300, Turbo Drive 400 *)
(* TD20 Classic Via Remote X1 Connector 9-way PLC interface*)
(* When serial interface is implemented, call Method M_Serial_IO after fb instantiation, in order to add the serial status *)
FUNCTION_BLOCK FB_PTM_TurboDrive EXTENDS FB_Pump
VAR_IN_OUT
END_VAR
VAR_INPUT
	i_xExtILKOk : BOOL; // Connect to external interlock logic, TRUE if not used.
END_VAR
VAR_OUTPUT
	{attribute 'pytmc' := '
    pv: 
	'}
	iq_stPtm	:	ST_LeyboldPTM;
END_VAR
VAR
	
	xRunOk	:	BOOL;
	tofRemoteDelay	:	TOF;
	
	
	(*IO*)
	i_xAtSpd AT%I*: BOOL; // Normaml operation when true
	i_xFaultNC AT%I*: BOOL; // Error Active when no Error is present
	q_RunDO AT%Q*: BOOL; // Start/Stop

END_VAR

(* Basic Turbo Control *)
(* This Function block provides basic turbo control for Leybold Turbo Drive 300, Turbo Drive 400 *)
(* TD20 Classic Via Remote X1 Connector 9-way PLC interface*)
(* M. Ghaly Jan. 2019 *)

(* Interlock Sum *)
iq_stPtm.xExtRunOk:= i_xExtILKOk;
xRunOk := iq_stPtm.xExtRunOk AND iq_stPtm.i_xNCError;

(* Basic pump supervisory section *)
IF xRunOk THEN
	q_RunDO := iq_stPTM.xRunSW;
ELSE
	iq_stPtm.xRunSW:=FALSE;
	q_RunDO:=FALSE;
END_IF

(*Pump States*)
IF (iq_stPtm.i_xFault) THEN
		iq_stPtm.eState := pumpFAULT;
		iq_stPtm.xRunSW:=FALSE;
		q_RunDO:=FALSE;
ELSIF (iq_stPtm.q_RunDO) AND (iq_stPtm.i_xAtSpd) THEN
		iq_stPtm.eState := pumpRUNNING;
ELSIF (iq_stPtm.q_RunDO) AND NOT (iq_stPtm.i_xAtSpd) THEN
		iq_stPtm.eState := pumpSTARTING; 
ELSIF NOT (iq_stPtm.q_RunDO) THEN
		iq_stPtm.eState := pumpSTOPPED;
ELSE 
	iq_stPtm.eState := pumpFAULT; 	
END_IF;
			

(*I/O soft mapping*)
ACT_IO();
// Log States and triggers
This^.ACT_Logger();

ACTION ACT_IO:
(*Inputs*)
iq_stPtm.i_xAtSpd := i_xAtSpd;
iq_stPtm.i_xNCError := i_xFaultNC;
iq_stPtm.i_xFault := NOT i_xFaultNC;



(*Outputs*)
iq_stPtm.q_RunDO := q_RunDO;
END_ACTION

ACTION ACT_Logger:
//STATE Logger  
// ILK logger
IF NOT i_xExtIlkOK AND ePrevState = pumpRUNNING THEN
 		fbLogger(sMsg:='Lost external interlock while pump was running.', eSevr:=TcEventSeverity.Critical);  	
END_IF


IF ePrevState <> iq_stPTM.eState THEN
	  CASE iq_stPTM.eState OF
		pumpFAULT:
			fbLogger(sMsg:='Pump Fault.', eSevr:=TcEventSeverity.Critical);
  		pumpSTOPPED:
			fbLogger(sMsg:='Pump stopped.', eSevr:=TcEventSeverity.Critical);
		pumpSTARTING:
			fbLogger(sMsg:='Pump starting.', eSevr:=TcEventSeverity.Info);
		pumpRUNNING:
			fbLogger(sMsg:='Pump running.', eSevr:=TcEventSeverity.Info);
	  END_CASE
	  ePrevState := iq_stPTM.eState;  
  END_IF
  
// Log Action
tAction(CLK:=  iq_stPTM.q_RunDO);
IF tAction.Q THEN fbLogger(sMsg:='Pump commanded to start', eSevr:=TcEventSeverity.Info); END_IF


// Log FAULT
tFault(CLK:= NOT iq_stPTM.i_xFault);
IF tFault.Q THEN fbLogger(sMsg:='Pump Lost Alarm OK bit', eSevr:=TcEventSeverity.Critical); END_IF
END_ACTION

METHOD PUBLIC M_Run : BOOL
VAR_INPUT
	run:bool; // set to true to run, false to stop;
END_VAR

this^.iq_stPtm.xRunSW := run;
END_METHOD

